SPLINE
SPL {X  -123.821, Y  +785.537, Z    +0.000, E1   -64.536, E3 +53300.374}
SPL {X  -153.467, Y  +737.853, Z    +0.000, E1   -51.757, E3 +53302.688}
SPL {X  -162.176, Y  +709.248, Z    +0.000, E1   -35.773, E3 +53301.714}
SPL {X  -164.888, Y  +691.368, Z    +0.000, E1   -20.174, E3 +53300.151}
SPL {X  -165.597, Y  +679.703, Z    +0.000, E1    -7.645, E3 +53300.327}
SPL {X  -165.650, Y  +673.520, Z    +0.000, E1    -0.048, E3 +53299.278}
SPL {X  -165.650, Y  +671.692, Z    +0.000, E1    +4.450, E3 +53298.845}
SPL {X  -165.650, Y  +667.743, Z    +0.000, E1   +15.617, E3 +53298.763}
SPL {X  -165.650, Y  +661.459, Z    +0.000, E1   +33.218, E3 +53298.343}
SPL {X  -165.650, Y  +653.296, Z    +0.000, E1   +51.333, E3 +53297.899}
SPL {X  -165.650, Y  +642.000, Z    +0.000, E1   +65.561, E3 +53297.111}
SPL {X  -165.650, Y  +619.979, Z    +0.000, E1   +79.465, E3 +53293.117}
SPL {X  -165.650, Y  +584.722, Z    +0.000, E1   +79.551, E3 +53302.408}
SPL {X  -165.650, Y  +560.326, Z    +0.000, E1   +78.360, E3 +53312.131}
SPL {X  -158.840, Y  +331.491, Z    +0.000, E1   +77.462, E3 +53394.706}
ENDSPLINE

SPLINE
SPL {X  -159.893, Y  +335.208, Z    +0.000, E1   +75.483, E3 +53415.441}
ENDSPLINE

SPLINE
SPL {X  -156.487, Y  +324.170, Z    +0.000, E1   +75.150, E3 +53424.822}
SPL {X  -142.256, Y  +293.629, Z    +0.000, E1   +77.020, E3 +53419.922}
ENDSPLINE

SPLINE
SPL {X  -142.811, Y  +294.566, Z    +0.000, E1   +75.668, E3 +53431.884}
ENDSPLINE

SPLINE
SPL {X  -141.646, Y  +292.615, Z    +0.000, E1   +74.702, E3 +53440.978}
SPL {X  -140.419, Y  +290.622, Z    +0.000, E1   +73.705, E3 +53449.821}
SPL {X  -136.008, Y  +283.940, Z    +0.000, E1   +73.594, E3 +53453.940}
SPL {X  -132.748, Y  +279.415, Z    +0.000, E1   +73.006, E3 +53459.996}
SPL {X  -129.007, Y  +274.590, Z    +0.000, E1   +72.484, E3 +53465.345}
SPL {X  -124.646, Y  +269.397, Z    +0.000, E1   +72.041, E3 +53470.093}
SPL {X  -111.023, Y  +255.562, Z    +0.000, E1   +75.772, E3 +53461.874}
SPL {X   -52.752, Y  +221.474, Z    +0.000, E1   +59.157, E3 +53591.126}
SPL {X   -49.901, Y  +220.545, Z    +0.000, E1   +56.696, E3 +53677.518}
ENDSPLINE

SPLINE
SPL {X  -127.117, Y  +272.287, Z    +0.000, E1   +62.713, E3 +53823.811}
SPL {X  -152.442, Y  +313.682, Z    +0.000, E1   +51.943, E3 +53828.043}
SPL {X  -159.925, Y  +335.326, Z    +0.000, E1   +41.361, E3 +53827.985}
SPL {X  -163.450, Y  +351.595, Z    +0.000, E1   +29.785, E3 +53827.096}
SPL {X  -165.127, Y  +365.342, Z    +0.000, E1   +17.250, E3 +53827.076}
SPL {X  -165.640, Y  +376.693, Z    +0.000, E1    +4.721, E3 +53826.649}
SPL {X  -165.650, Y  +380.500, Z    +0.000, E1    -0.000, E3 +53825.800}
SPL {X  -165.650, Y  +383.262, Z    +0.000, E1    -6.645, E3 +53825.329}
SPL {X  -165.650, Y  +388.390, Z    +0.000, E1   -21.508, E3 +53825.117}
SPL {X  -165.650, Y  +393.439, Z    +0.000, E1   -35.398, E3 +53824.685}
SPL {X  -165.650, Y  +400.610, Z    +0.000, E1   -50.510, E3 +53824.422}
SPL {X  -165.650, Y  +414.376, Z    +0.000, E1   -68.098, E3 +53822.456}
SPL {X  -165.650, Y  +468.582, Z    +0.000, E1   -78.237, E3 +53831.226}
SPL {X  -158.306, Y  +724.277, Z    +0.000, E1   -77.461, E3 +53921.667}
ENDSPLINE

SPLINE
SPL {X  -160.145, Y  +717.851, Z    +0.000, E1   -75.386, E3 +53942.181}
ENDSPLINE

SPLINE
SPL {X  -157.156, Y  +727.862, Z    +0.000, E1   -75.175, E3 +53949.653}
SPL {X  -154.068, Y  +736.353, Z    +0.000, E1   -74.906, E3 +53956.828}
SPL {X  -149.738, Y  +746.340, Z    +0.000, E1   -74.451, E3 +53966.515}
SPL {X  -145.204, Y  +755.223, Z    +0.000, E1   -74.188, E3 +53973.242}
SPL {X  -142.724, Y  +759.583, Z    +0.000, E1   -73.634, E3 +53980.061}
SPL {X  -138.277, Y  +766.711, Z    +0.000, E1   -73.303, E3 +53986.192}
SPL {X  -134.662, Y  +771.969, Z    +0.000, E1   -72.884, E3 +53991.634}
SPL {X  -131.459, Y  +776.289, Z    +0.000, E1   -72.475, E3 +53996.301}
SPL {X  -128.771, Y  +779.702, Z    +0.000, E1   -71.875, E3 +54001.248}
SPL {X  -125.267, Y  +783.889, Z    +0.000, E1   -71.674, E3 +54004.360}
SPL {X  -119.086, Y  +790.645, Z    +0.000, E1   -72.931, E3 +54002.647}
SPL {X   -51.449, Y  +832.958, Z    +0.000, E1   -57.230, E3 +54160.167}
ENDSPLINE

SPLINE
SPL {X  -123.821, Y  +785.537, Z    +0.000, E1   -64.536, E3 +54361.912}
SPL {X  -153.467, Y  +737.853, Z    +0.000, E1   -51.757, E3 +54364.227}
SPL {X  -162.176, Y  +709.248, Z    +0.000, E1   -35.773, E3 +54363.252}
SPL {X  -164.888, Y  +691.368, Z    +0.000, E1   -20.174, E3 +54361.690}
SPL {X  -165.597, Y  +679.703, Z    +0.000, E1    -7.645, E3 +54361.865}
SPL {X  -165.650, Y  +673.520, Z    +0.000, E1    -0.048, E3 +54360.817}
SPL {X  -165.650, Y  +671.692, Z    +0.000, E1    +4.450, E3 +54360.383}
SPL {X  -165.650, Y  +667.743, Z    +0.000, E1   +15.617, E3 +54360.301}
SPL {X  -165.650, Y  +662.891, Z    +0.000, E1   +29.740, E3 +54359.819}
SPL {X  -165.650, Y  +655.319, Z    +0.000, E1   +47.265, E3 +54359.668}
SPL {X  -165.650, Y  +642.000, Z    +0.000, E1   +65.561, E3 +54358.649}
SPL {X  -165.650, Y  +619.979, Z    +0.000, E1   +79.465, E3 +54354.656}
SPL {X  -165.650, Y  +569.632, Z    +0.000, E1   +78.783, E3 +54369.935}
SPL {X  -160.258, Y  +336.579, Z    +0.000, E1   +78.314, E3 +54445.191}
SPL {X  -159.618, Y  +334.207, Z    +0.000, E1   +75.622, E3 +54476.005}
SPL {X  -156.487, Y  +324.170, Z    +0.000, E1   +75.150, E3 +54486.360}
SPL {X  -142.256, Y  +293.629, Z    +0.000, E1   +77.020, E3 +54481.460}
ENDSPLINE

SPLINE
SPL {X  -142.811, Y  +294.566, Z    +0.000, E1   +75.668, E3 +54493.422}
ENDSPLINE

SPLINE
SPL {X  -141.646, Y  +292.615, Z    +0.000, E1   +74.702, E3 +54502.516}
SPL {X  -140.419, Y  +290.622, Z    +0.000, E1   +73.705, E3 +54511.359}
SPL {X  -136.008, Y  +283.940, Z    +0.000, E1   +73.594, E3 +54515.478}
SPL {X  -132.748, Y  +279.415, Z    +0.000, E1   +73.006, E3 +54521.534}
SPL {X  -129.007, Y  +274.590, Z    +0.000, E1   +72.484, E3 +54526.883}
SPL {X  -125.914, Y  +270.864, Z    +0.000, E1   +72.144, E3 +54530.375}
SPL {X  -123.729, Y  +268.359, Z    +0.000, E1   +71.932, E3 +54532.547}
SPL {X  -111.023, Y  +255.562, Z    +0.000, E1   +75.772, E3 +54523.413}
SPL {X   -49.289, Y  +220.353, Z    +0.000, E1   +56.690, E3 +54716.128}
ENDSPLINE

SPLINE
SPL {X  -127.117, Y  +272.287, Z    +0.000, E1   +62.713, E3 +54885.350}
SPL {X  -152.442, Y  +313.682, Z    +0.000, E1   +51.943, E3 +54889.581}
SPL {X  -159.925, Y  +335.326, Z    +0.000, E1   +41.361, E3 +54889.523}
SPL {X  -163.450, Y  +351.595, Z    +0.000, E1   +29.785, E3 +54888.635}
SPL {X  -165.127, Y  +365.342, Z    +0.000, E1   +17.250, E3 +54888.615}
SPL {X  -165.640, Y  +376.693, Z    +0.000, E1    +4.721, E3 +54888.188}
SPL {X  -165.650, Y  +380.500, Z    +0.000, E1    -0.000, E3 +54887.339}
SPL {X  -165.650, Y  +382.123, Z    +0.000, E1    -3.912, E3 +54886.966}
SPL {X  -165.650, Y  +387.069, Z    +0.000, E1   -17.420, E3 +54886.677}
SPL {X  -165.650, Y  +393.439, Z    +0.000, E1   -35.398, E3 +54886.223}
SPL {X  -165.650, Y  +400.610, Z    +0.000, E1   -50.510, E3 +54885.961}
SPL {X  -165.650, Y  +414.376, Z    +0.000, E1   -68.098, E3 +54883.994}
SPL {X  -165.650, Y  +468.582, Z    +0.000, E1   -78.237, E3 +54892.765}
SPL {X  -160.244, Y  +717.475, Z    +0.000, E1   -78.917, E3 +54965.322}
SPL {X  -159.651, Y  +719.676, Z    +0.000, E1   -75.661, E3 +55001.709}
SPL {X  -157.156, Y  +727.862, Z    +0.000, E1   -75.175, E3 +55011.191}
SPL {X  -152.814, Y  +739.436, Z    +0.000, E1   -74.813, E3 +55021.045}
SPL {X  -148.754, Y  +748.385, Z    +0.000, E1   -74.281, E3 +55030.487}
SPL {X  -144.163, Y  +757.090, Z    +0.000, E1   -74.033, E3 +55037.146}
SPL {X  -139.284, Y  +765.165, Z    +0.000, E1   -73.322, E3 +55046.841}
SPL {X  -134.662, Y  +771.969, Z    +0.000, E1   -72.884, E3 +55053.173}
SPL {X  -131.459, Y  +776.289, Z    +0.000, E1   -72.475, E3 +55057.840}
SPL {X  -128.771, Y  +779.702, Z    +0.000, E1   -71.875, E3 +55062.786}
SPL {X  -124.506, Y  +784.762, Z    +0.000, E1   -71.815, E3 +55065.675}
SPL {X  -112.958, Y  +796.663, Z    +0.000, E1   -74.119, E3 +55062.378}
SPL {X   -54.274, Y  +832.006, Z    +0.000, E1   -58.502, E3 +55194.398}
SPL {X   -50.797, Y  +833.169, Z    +0.000, E1   -57.000, E3 +55289.747}
ENDSPLINE

SPLINE
SPL {X  -113.713, Y  +795.955, Z    +0.000, E1   -65.735, E3 +55420.624}
SPL {X  -131.116, Y  +776.736, Z    +0.000, E1   -63.149, E3 +55425.154}
SPL {X  -153.467, Y  +737.853, Z    +0.000, E1   -51.757, E3 +55425.765}
SPL {X  -162.176, Y  +709.248, Z    +0.000, E1   -35.773, E3 +55424.791}
SPL {X  -164.888, Y  +691.368, Z    +0.000, E1   -20.174, E3 +55423.228}
SPL {X  -165.597, Y  +679.703, Z    +0.000, E1    -7.645, E3 +55423.403}
SPL {X  -165.650, Y  +673.520, Z    +0.000, E1    -0.048, E3 +55422.355}
SPL {X  -165.650, Y  +671.692, Z    +0.000, E1    +4.450, E3 +55421.922}
SPL {X  -165.650, Y  +667.743, Z    +0.000, E1   +15.617, E3 +55421.840}
SPL {X  -165.650, Y  +662.891, Z    +0.000, E1   +29.740, E3 +55421.358}
SPL {X  -165.650, Y  +655.319, Z    +0.000, E1   +47.265, E3 +55421.206}
SPL {X  -165.650, Y  +642.000, Z    +0.000, E1   +65.561, E3 +55420.188}
SPL {X  -165.650, Y  +619.979, Z    +0.000, E1   +79.465, E3 +55416.194}
SPL {X  -165.650, Y  +569.632, Z    +0.000, E1   +78.783, E3 +55431.473}
SPL {X  -158.840, Y  +331.491, Z    +0.000, E1   +77.462, E3 +55517.783}
ENDSPLINE

SPLINE
SPL {X  -159.893, Y  +335.208, Z    +0.000, E1   +75.483, E3 +55538.518}
ENDSPLINE

SPLINE
SPL {X  -156.487, Y  +324.170, Z    +0.000, E1   +75.150, E3 +55547.899}
SPL {X  -142.256, Y  +293.629, Z    +0.000, E1   +77.020, E3 +55542.999}
ENDSPLINE

SPLINE
SPL {X  -142.811, Y  +294.566, Z    +0.000, E1   +75.668, E3 +55554.961}
ENDSPLINE

SPLINE
SPL {X  -141.646, Y  +292.615, Z    +0.000, E1   +74.702, E3 +55564.055}
SPL {X  -140.419, Y  +290.622, Z    +0.000, E1   +73.705, E3 +55572.898}
SPL {X  -135.839, Y  +283.697, Z    +0.000, E1   +73.388, E3 +55578.636}
SPL {X  -131.336, Y  +277.551, Z    +0.000, E1   +72.879, E3 +55584.888}
SPL {X  -126.848, Y  +271.966, Z    +0.000, E1   +72.322, E3 +55590.617}
SPL {X  -123.729, Y  +268.359, Z    +0.000, E1   +71.932, E3 +55594.085}
SPL {X  -111.023, Y  +255.562, Z    +0.000, E1   +75.772, E3 +55584.951}
SPL {X   -52.752, Y  +221.474, Z    +0.000, E1   +59.157, E3 +55714.203}
SPL {X   -49.901, Y  +220.545, Z    +0.000, E1   +56.696, E3 +55800.595}
ENDSPLINE

SPLINE
SPL {X  -127.117, Y  +272.287, Z    +0.000, E1   +62.713, E3 +55946.888}
SPL {X  -152.442, Y  +313.682, Z    +0.000, E1   +51.943, E3 +55951.120}
SPL {X  -162.319, Y  +345.447, Z    +0.000, E1   +34.671, E3 +55950.545}
SPL {X  -165.127, Y  +365.342, Z    +0.000, E1   +17.250, E3 +55950.153}
SPL {X  -165.640, Y  +376.693, Z    +0.000, E1    +4.721, E3 +55949.726}
SPL {X  -165.650, Y  +380.500, Z    +0.000, E1    -0.000, E3 +55948.877}
SPL {X  -165.650, Y  +383.262, Z    +0.000, E1    -6.645, E3 +55948.406}
SPL {X  -165.650, Y  +388.390, Z    +0.000, E1   -21.508, E3 +55948.194}
SPL {X  -165.650, Y  +393.439, Z    +0.000, E1   -35.398, E3 +55947.762}
SPL {X  -165.650, Y  +400.610, Z    +0.000, E1   -50.510, E3 +55947.499}
SPL {X  -165.650, Y  +414.376, Z    +0.000, E1   -68.098, E3 +55945.533}
SPL {X  -165.650, Y  +468.582, Z    +0.000, E1   -78.237, E3 +55954.303}
SPL {X  -158.306, Y  +724.277, Z    +0.000, E1   -77.461, E3 +56044.744}
ENDSPLINE

SPLINE
SPL {X  -160.145, Y  +717.851, Z    +0.000, E1   -75.386, E3 +56065.258}
ENDSPLINE

SPLINE
SPL {X  -157.156, Y  +727.862, Z    +0.000, E1   -75.175, E3 +56072.730}
SPL {X  -152.814, Y  +739.436, Z    +0.000, E1   -74.813, E3 +56082.583}
SPL {X  -148.754, Y  +748.385, Z    +0.000, E1   -74.281, E3 +56092.026}
SPL {X  -144.163, Y  +757.090, Z    +0.000, E1   -74.033, E3 +56098.685}
SPL {X  -139.284, Y  +765.165, Z    +0.000, E1   -73.322, E3 +56108.379}
SPL {X  -134.662, Y  +771.969, Z    +0.000, E1   -72.884, E3 +56114.711}
SPL {X  -131.459, Y  +776.289, Z    +0.000, E1   -72.475, E3 +56119.378}
SPL {X  -127.605, Y  +781.126, Z    +0.000, E1   -71.922, E3 +56124.822}
SPL {X  -124.773, Y  +784.457, Z    +0.000, E1   -71.383, E3 +56128.870}
SPL {X  -119.086, Y  +790.645, Z    +0.000, E1   -72.931, E3 +56125.724}
SPL {X   -51.449, Y  +832.958, Z    +0.000, E1   -57.230, E3 +56283.244}
ENDSPLINE

SPLINE
SPL {X  -123.821, Y  +785.537, Z    +0.000, E1   -64.536, E3 +56484.989}
SPL {X  -153.467, Y  +737.853, Z    +0.000, E1   -51.757, E3 +56487.304}
SPL {X  -162.176, Y  +709.248, Z    +0.000, E1   -35.773, E3 +56486.329}
SPL {X  -164.888, Y  +691.368, Z    +0.000, E1   -20.174, E3 +56484.767}
SPL {X  -165.597, Y  +679.703, Z    +0.000, E1    -7.645, E3 +56484.942}
SPL {X  -165.650, Y  +673.520, Z    +0.000, E1    -0.048, E3 +56483.894}
SPL {X  -165.650, Y  +671.692, Z    +0.000, E1    +4.450, E3 +56483.460}
SPL {X  -165.650, Y  +667.743, Z    +0.000, E1   +15.617, E3 +56483.378}
SPL {X  -165.650, Y  +661.459, Z    +0.000, E1   +33.218, E3 +56482.959}
SPL {X  -165.650, Y  +653.296, Z    +0.000, E1   +51.333, E3 +56482.514}
SPL {X  -165.650, Y  +642.000, Z    +0.000, E1   +65.561, E3 +56481.726}
SPL {X  -165.650, Y  +619.979, Z    +0.000, E1   +79.465, E3 +56477.733}
SPL {X  -165.650, Y  +584.722, Z    +0.000, E1   +79.551, E3 +56487.023}
SPL {X  -165.650, Y  +560.326, Z    +0.000, E1   +78.360, E3 +56496.746}
SPL {X  -158.840, Y  +331.491, Z    +0.000, E1   +77.462, E3 +56579.322}
ENDSPLINE

SPLINE
SPL {X  -159.893, Y  +335.208, Z    +0.000, E1   +75.483, E3 +56600.056}
ENDSPLINE

SPLINE
SPL {X  -156.487, Y  +324.170, Z    +0.000, E1   +75.150, E3 +56609.437}
SPL {X  -142.256, Y  +293.629, Z    +0.000, E1   +77.020, E3 +56604.537}
ENDSPLINE

SPLINE
SPL {X  -142.811, Y  +294.566, Z    +0.000, E1   +75.668, E3 +56616.499}
ENDSPLINE

SPLINE
SPL {X  -141.646, Y  +292.615, Z    +0.000, E1   +74.702, E3 +56625.593}
SPL {X  -140.419, Y  +290.622, Z    +0.000, E1   +73.705, E3 +56634.436}
SPL {X  -136.008, Y  +283.940, Z    +0.000, E1   +73.594, E3 +56638.555}
SPL {X  -132.748, Y  +279.415, Z    +0.000, E1   +73.006, E3 +56644.611}
SPL {X  -129.007, Y  +274.590, Z    +0.000, E1   +72.484, E3 +56649.960}
SPL {X  -124.646, Y  +269.397, Z    +0.000, E1   +72.041, E3 +56654.708}
SPL {X  -111.023, Y  +255.562, Z    +0.000, E1   +75.772, E3 +56646.490}
SPL {X   -52.752, Y  +221.474, Z    +0.000, E1   +59.157, E3 +56775.741}
SPL {X   -49.901, Y  +220.545, Z    +0.000, E1   +56.696, E3 +56862.134}
ENDSPLINE

SPLINE
SPL {X  -127.117, Y  +272.287, Z    +0.000, E1   +62.713, E3 +57008.427}
SPL {X  -152.442, Y  +313.682, Z    +0.000, E1   +51.943, E3 +57012.658}
SPL {X  -159.925, Y  +335.326, Z    +0.000, E1   +41.361, E3 +57012.600}
SPL {X  -163.450, Y  +351.595, Z    +0.000, E1   +29.785, E3 +57011.712}
SPL {X  -165.127, Y  +365.342, Z    +0.000, E1   +17.250, E3 +57011.692}
SPL {X  -165.640, Y  +376.693, Z    +0.000, E1    +4.721, E3 +57011.265}
SPL {X  -165.650, Y  +380.500, Z    +0.000, E1    -0.000, E3 +57010.416}
SPL {X  -165.650, Y  +383.262, Z    +0.000, E1    -6.645, E3 +57009.945}
SPL {X  -165.650, Y  +388.390, Z    +0.000, E1   -21.508, E3 +57009.733}
SPL {X  -165.650, Y  +393.439, Z    +0.000, E1   -35.398, E3 +57009.300}
SPL {X  -165.650, Y  +400.610, Z    +0.000, E1   -50.510, E3 +57009.038}
SPL {X  -165.650, Y  +414.376, Z    +0.000, E1   -68.098, E3 +57007.071}
SPL {X  -165.650, Y  +468.582, Z    +0.000, E1   -78.237, E3 +57015.841}
SPL {X  -158.306, Y  +724.277, Z    +0.000, E1   -77.461, E3 +57106.283}
ENDSPLINE

SPLINE
SPL {X  -160.145, Y  +717.851, Z    +0.000, E1   -75.386, E3 +57126.796}
ENDSPLINE

SPLINE
SPL {X  -157.156, Y  +727.862, Z    +0.000, E1   -75.175, E3 +57134.268}
SPL {X  -152.814, Y  +739.436, Z    +0.000, E1   -74.813, E3 +57144.122}
SPL {X  -147.104, Y  +751.659, Z    +0.000, E1   -74.255, E3 +57155.566}
SPL {X  -141.453, Y  +761.704, Z    +0.000, E1   -73.638, E3 +57165.779}
SPL {X  -135.914, Y  +770.196, Z    +0.000, E1   -72.974, E3 +57174.841}
SPL {X  -131.459, Y  +776.289, Z    +0.000, E1   -72.475, E3 +57180.917}
SPL {X  -127.605, Y  +781.126, Z    +0.000, E1   -71.922, E3 +57186.361}
SPL {X  -124.773, Y  +784.457, Z    +0.000, E1   -71.383, E3 +57190.408}
SPL {X  -119.086, Y  +790.645, Z    +0.000, E1   -72.931, E3 +57187.262}
SPL {X   -51.449, Y  +832.958, Z    +0.000, E1   -57.230, E3 +57344.782}
ENDSPLINE

SPLINE
SPL {X  -113.713, Y  +795.955, Z    +0.000, E1   -65.735, E3 +57543.701}
SPL {X  -131.116, Y  +776.736, Z    +0.000, E1   -63.149, E3 +57548.231}
SPL {X  -153.467, Y  +737.853, Z    +0.000, E1   -51.757, E3 +57548.842}
SPL {X  -161.000, Y  +714.475, Z    +0.000, E1   -39.424, E3 +57548.315}
SPL {X  -164.534, Y  +694.695, Z    +0.000, E1   -23.511, E3 +57546.605}
SPL {X  -165.597, Y  +679.703, Z    +0.000, E1    -7.645, E3 +57546.480}
SPL {X  -165.650, Y  +673.520, Z    +0.000, E1    -0.048, E3 +57545.432}
SPL {X  -165.650, Y  +671.692, Z    +0.000, E1    +4.450, E3 +57544.999}
SPL {X  -165.650, Y  +667.743, Z    +0.000, E1   +15.617, E3 +57544.917}
SPL {X  -165.650, Y  +661.459, Z    +0.000, E1   +33.218, E3 +57544.497}
SPL {X  -165.650, Y  +650.834, Z    +0.000, E1   +55.143, E3 +57543.885}
SPL {X  -165.650, Y  +639.785, Z    +0.000, E1   +67.512, E3 +57543.102}
SPL {X  -165.650, Y  +619.979, Z    +0.000, E1   +79.465, E3 +57539.271}
SPL {X  -165.650, Y  +584.722, Z    +0.000, E1   +79.551, E3 +57548.562}
SPL {X  -165.650, Y  +560.326, Z    +0.000, E1   +78.360, E3 +57558.284}
SPL {X  -160.258, Y  +336.579, Z    +0.000, E1   +78.314, E3 +57629.806}
SPL {X  -159.618, Y  +334.207, Z    +0.000, E1   +75.622, E3 +57660.620}
SPL {X  -156.487, Y  +324.170, Z    +0.000, E1   +75.150, E3 +57670.976}
SPL {X  -142.256, Y  +293.629, Z    +0.000, E1   +77.020, E3 +57666.076}
ENDSPLINE

SPLINE
SPL {X  -142.811, Y  +294.566, Z    +0.000, E1   +75.668, E3 +57678.038}
ENDSPLINE

SPLINE
SPL {X  -141.646, Y  +292.615, Z    +0.000, E1   +74.702, E3 +57687.131}
SPL {X  -140.419, Y  +290.622, Z    +0.000, E1   +73.705, E3 +57695.975}
SPL {X  -135.839, Y  +283.697, Z    +0.000, E1   +73.388, E3 +57701.713}
SPL {X  -131.903, Y  +278.292, Z    +0.000, E1   +73.096, E3 +57706.202}
SPL {X  -129.007, Y  +274.590, Z    +0.000, E1   +72.484, E3 +57711.498}
SPL {X  -124.646, Y  +269.397, Z    +0.000, E1   +72.041, E3 +57716.247}
SPL {X  -111.023, Y  +255.562, Z    +0.000, E1   +75.772, E3 +57708.028}
SPL {X   -49.289, Y  +220.353, Z    +0.000, E1   +56.690, E3 +57900.743}
ENDSPLINE

SPLINE
SPL {X  -127.117, Y  +272.287, Z    +0.000, E1   +62.713, E3 +58069.965}
SPL {X  -152.442, Y  +313.682, Z    +0.000, E1   +51.943, E3 +58074.197}
SPL {X  -159.925, Y  +335.326, Z    +0.000, E1   +41.361, E3 +58074.139}
SPL {X  -163.450, Y  +351.595, Z    +0.000, E1   +29.785, E3 +58073.250}
SPL {X  -165.127, Y  +365.342, Z    +0.000, E1   +17.250, E3 +58073.230}
SPL {X  -165.640, Y  +376.693, Z    +0.000, E1    +4.721, E3 +58072.803}
SPL {X  -165.650, Y  +380.500, Z    +0.000, E1    -0.000, E3 +58071.954}
SPL {X  -165.650, Y  +382.123, Z    +0.000, E1    -3.912, E3 +58071.581}
SPL {X  -165.650, Y  +387.069, Z    +0.000, E1   -17.420, E3 +58071.293}
SPL {X  -165.650, Y  +393.439, Z    +0.000, E1   -35.398, E3 +58070.839}
SPL {X  -165.650, Y  +400.610, Z    +0.000, E1   -50.510, E3 +58070.576}
SPL {X  -165.650, Y  +414.376, Z    +0.000, E1   -68.098, E3 +58068.610}
SPL {X  -165.650, Y  +468.582, Z    +0.000, E1   -78.237, E3 +58077.380}
SPL {X  -158.306, Y  +724.277, Z    +0.000, E1   -77.461, E3 +58167.821}
ENDSPLINE

SPLINE
SPL {X  -160.145, Y  +717.851, Z    +0.000, E1   -75.386, E3 +58188.335}
ENDSPLINE

SPLINE
SPL {X  -157.156, Y  +727.862, Z    +0.000, E1   -75.175, E3 +58195.807}
SPL {X  -154.068, Y  +736.353, Z    +0.000, E1   -74.906, E3 +58202.981}
SPL {X  -149.738, Y  +746.340, Z    +0.000, E1   -74.451, E3 +58212.669}
SPL {X  -145.204, Y  +755.223, Z    +0.000, E1   -74.188, E3 +58219.395}
SPL {X  -142.724, Y  +759.583, Z    +0.000, E1   -73.634, E3 +58226.215}
SPL {X  -138.277, Y  +766.711, Z    +0.000, E1   -73.303, E3 +58232.346}
SPL {X  -134.662, Y  +771.969, Z    +0.000, E1   -72.884, E3 +58237.788}
SPL {X  -131.459, Y  +776.289, Z    +0.000, E1   -72.475, E3 +58242.455}
SPL {X  -128.771, Y  +779.702, Z    +0.000, E1   -71.875, E3 +58247.402}
SPL {X  -124.506, Y  +784.762, Z    +0.000, E1   -71.815, E3 +58250.290}
SPL {X  -112.958, Y  +796.663, Z    +0.000, E1   -74.119, E3 +58246.994}
SPL {X   -51.449, Y  +832.958, Z    +0.000, E1   -57.230, E3 +58406.321}
ENDSPLINE

SPLINE
SPL {X  -123.821, Y  +785.537, Z    +0.000, E1   -64.536, E3 +58608.066}
SPL {X  -153.467, Y  +737.853, Z    +0.000, E1   -51.757, E3 +58610.381}
SPL {X  -161.000, Y  +714.475, Z    +0.000, E1   -39.424, E3 +58609.853}
SPL {X  -164.534, Y  +694.695, Z    +0.000, E1   -23.511, E3 +58608.143}
SPL {X  -165.597, Y  +679.703, Z    +0.000, E1    -7.645, E3 +58608.019}
SPL {X  -165.650, Y  +673.520, Z    +0.000, E1    -0.048, E3 +58606.971}
SPL {X  -165.650, Y  +671.692, Z    +0.000, E1    +4.450, E3 +58606.537}
SPL {X  -165.650, Y  +667.743, Z    +0.000, E1   +15.617, E3 +58606.455}
SPL {X  -165.650, Y  +662.891, Z    +0.000, E1   +29.740, E3 +58605.973}
SPL {X  -165.650, Y  +655.319, Z    +0.000, E1   +47.265, E3 +58605.822}
SPL {X  -165.650, Y  +642.000, Z    +0.000, E1   +65.561, E3 +58604.803}
SPL {X  -165.650, Y  +619.979, Z    +0.000, E1   +79.465, E3 +58600.810}
SPL {X  -165.650, Y  +569.632, Z    +0.000, E1   +78.783, E3 +58616.088}
SPL {X  -158.840, Y  +331.491, Z    +0.000, E1   +77.462, E3 +58702.398}
ENDSPLINE

SPLINE
SPL {X  -159.893, Y  +335.208, Z    +0.000, E1   +75.483, E3 +58723.133}
ENDSPLINE

SPLINE
SPL {X  -156.487, Y  +324.170, Z    +0.000, E1   +75.150, E3 +58732.514}
SPL {X  -142.256, Y  +293.629, Z    +0.000, E1   +77.020, E3 +58727.614}
ENDSPLINE

SPLINE
SPL {X  -142.811, Y  +294.566, Z    +0.000, E1   +75.668, E3 +58739.576}
ENDSPLINE

SPLINE
SPL {X  -141.646, Y  +292.615, Z    +0.000, E1   +74.702, E3 +58748.670}
SPL {X  -140.419, Y  +290.622, Z    +0.000, E1   +73.705, E3 +58757.513}
SPL {X  -136.008, Y  +283.940, Z    +0.000, E1   +73.594, E3 +58761.632}
SPL {X  -132.748, Y  +279.415, Z    +0.000, E1   +73.006, E3 +58767.688}
SPL {X  -129.007, Y  +274.590, Z    +0.000, E1   +72.484, E3 +58773.037}
SPL {X  -125.914, Y  +270.864, Z    +0.000, E1   +72.144, E3 +58776.528}
SPL {X  -123.729, Y  +268.359, Z    +0.000, E1   +71.932, E3 +58778.701}
SPL {X  -111.023, Y  +255.562, Z    +0.000, E1   +75.772, E3 +58769.567}
SPL {X   -52.752, Y  +221.474, Z    +0.000, E1   +59.157, E3 +58898.818}
SPL {X   -49.901, Y  +220.545, Z    +0.000, E1   +56.696, E3 +58985.211}
ENDSPLINE

SPLINE
SPL {X  -127.117, Y  +272.287, Z    +0.000, E1   +62.713, E3 +59131.503}
SPL {X  -152.442, Y  +313.682, Z    +0.000, E1   +51.943, E3 +59135.735}
SPL {X  -162.319, Y  +345.447, Z    +0.000, E1   +34.671, E3 +59135.161}
SPL {X  -165.127, Y  +365.342, Z    +0.000, E1   +17.250, E3 +59134.769}
SPL {X  -165.640, Y  +376.693, Z    +0.000, E1    +4.721, E3 +59134.342}
SPL {X  -165.650, Y  +380.500, Z    +0.000, E1    -0.000, E3 +59133.493}
SPL {X  -165.650, Y  +382.123, Z    +0.000, E1    -3.912, E3 +59133.120}
SPL {X  -165.650, Y  +387.069, Z    +0.000, E1   -17.420, E3 +59132.831}
SPL {X  -165.650, Y  +393.439, Z    +0.000, E1   -35.398, E3 +59132.377}
SPL {X  -165.650, Y  +400.610, Z    +0.000, E1   -50.510, E3 +59132.115}
SPL {X  -165.650, Y  +414.376, Z    +0.000, E1   -68.098, E3 +59130.148}
SPL {X  -165.650, Y  +468.582, Z    +0.000, E1   -78.237, E3 +59138.918}
SPL {X  -158.306, Y  +724.277, Z    +0.000, E1   -77.461, E3 +59229.360}
ENDSPLINE

SPLINE
SPL {X  -160.145, Y  +717.851, Z    +0.000, E1   -75.386, E3 +59249.873}
ENDSPLINE

SPLINE
SPL {X  -157.156, Y  +727.862, Z    +0.000, E1   -75.175, E3 +59257.345}
SPL {X  -154.068, Y  +736.353, Z    +0.000, E1   -74.906, E3 +59264.520}
SPL {X  -149.738, Y  +746.340, Z    +0.000, E1   -74.451, E3 +59274.208}
SPL {X  -144.163, Y  +757.090, Z    +0.000, E1   -74.033, E3 +59283.300}
SPL {X  -139.284, Y  +765.165, Z    +0.000, E1   -73.322, E3 +59292.995}
SPL {X  -134.662, Y  +771.969, Z    +0.000, E1   -72.884, E3 +59299.326}
SPL {X  -131.459, Y  +776.289, Z    +0.000, E1   -72.475, E3 +59303.994}
SPL {X  -127.605, Y  +781.126, Z    +0.000, E1   -71.922, E3 +59309.438}
SPL {X  -124.773, Y  +784.457, Z    +0.000, E1   -71.383, E3 +59313.485}
SPL {X  -119.086, Y  +790.645, Z    +0.000, E1   -72.931, E3 +59310.339}
SPL {X   -51.449, Y  +832.958, Z    +0.000, E1   -57.230, E3 +59467.859}
ENDSPLINE

SPLINE
SPL {X  -123.821, Y  +785.537, Z    +0.000, E1   -64.536, E3 +59669.604}
SPL {X  -153.467, Y  +737.853, Z    +0.000, E1   -51.757, E3 +59671.919}
SPL {X  -161.000, Y  +714.475, Z    +0.000, E1   -39.424, E3 +59671.392}
SPL {X  -164.534, Y  +694.695, Z    +0.000, E1   -23.511, E3 +59669.682}
SPL {X  -165.597, Y  +679.703, Z    +0.000, E1    -7.645, E3 +59669.557}
SPL {X  -165.650, Y  +673.520, Z    +0.000, E1    -0.048, E3 +59668.509}
SPL {X  -165.650, Y  +671.692, Z    +0.000, E1    +4.450, E3 +59668.076}
SPL {X  -165.650, Y  +667.743, Z    +0.000, E1   +15.617, E3 +59667.994}
SPL {X  -165.650, Y  +662.891, Z    +0.000, E1   +29.740, E3 +59667.511}
SPL {X  -165.650, Y  +655.319, Z    +0.000, E1   +47.265, E3 +59667.360}
SPL {X  -165.650, Y  +642.000, Z    +0.000, E1   +65.561, E3 +59666.341}
SPL {X  -165.650, Y  +619.979, Z    +0.000, E1   +79.465, E3 +59662.348}
SPL {X  -165.650, Y  +569.632, Z    +0.000, E1   +78.783, E3 +59677.627}
SPL {X  -160.258, Y  +336.579, Z    +0.000, E1   +78.314, E3 +59752.883}
SPL {X  -159.618, Y  +334.207, Z    +0.000, E1   +75.622, E3 +59783.697}
SPL {X  -156.487, Y  +324.170, Z    +0.000, E1   +75.150, E3 +59794.053}
SPL {X  -142.256, Y  +293.629, Z    +0.000, E1   +77.020, E3 +59789.152}
ENDSPLINE

SPLINE
SPL {X  -142.811, Y  +294.566, Z    +0.000, E1   +75.668, E3 +59801.115}
ENDSPLINE

SPLINE
SPL {X  -141.646, Y  +292.615, Z    +0.000, E1   +74.702, E3 +59810.208}
SPL {X  -140.419, Y  +290.622, Z    +0.000, E1   +73.705, E3 +59819.052}
SPL {X  -135.839, Y  +283.697, Z    +0.000, E1   +73.388, E3 +59824.790}
SPL {X  -131.336, Y  +277.551, Z    +0.000, E1   +72.879, E3 +59831.042}
SPL {X  -126.848, Y  +271.966, Z    +0.000, E1   +72.322, E3 +59836.770}
SPL {X  -123.729, Y  +268.359, Z    +0.000, E1   +71.932, E3 +59840.239}
SPL {X  -111.023, Y  +255.562, Z    +0.000, E1   +75.772, E3 +59831.105}
SPL {X   -49.289, Y  +220.353, Z    +0.000, E1   +56.690, E3 +60023.820}
ENDSPLINE

SPLINE
SPL {X  -127.117, Y  +272.287, Z    +0.000, E1   +62.713, E3 +60193.042}
SPL {X  -152.442, Y  +313.682, Z    +0.000, E1   +51.943, E3 +60197.274}
SPL {X  -159.925, Y  +335.326, Z    +0.000, E1   +41.361, E3 +60197.216}
SPL {X  -163.450, Y  +351.595, Z    +0.000, E1   +29.785, E3 +60196.327}
SPL {X  -165.127, Y  +365.342, Z    +0.000, E1   +17.250, E3 +60196.307}
SPL {X  -165.640, Y  +376.693, Z    +0.000, E1    +4.721, E3 +60195.880}
SPL {X  -165.650, Y  +380.500, Z    +0.000, E1    -0.000, E3 +60195.031}
SPL {X  -165.650, Y  +382.123, Z    +0.000, E1    -3.912, E3 +60194.658}
SPL {X  -165.650, Y  +387.069, Z    +0.000, E1   -17.420, E3 +60194.370}
SPL {X  -165.650, Y  +393.439, Z    +0.000, E1   -35.398, E3 +60193.915}
SPL {X  -165.650, Y  +400.610, Z    +0.000, E1   -50.510, E3 +60193.653}
SPL {X  -165.650, Y  +414.376, Z    +0.000, E1   -68.098, E3 +60191.687}
SPL {X  -165.650, Y  +468.582, Z    +0.000, E1   -78.237, E3 +60200.457}
SPL {X  -158.306, Y  +724.277, Z    +0.000, E1   -77.461, E3 +60290.898}
ENDSPLINE

SPLINE
SPL {X  -160.145, Y  +717.851, Z    +0.000, E1   -75.386, E3 +60311.412}
ENDSPLINE

SPLINE
SPL {X  -157.156, Y  +727.862, Z    +0.000, E1   -75.175, E3 +60318.884}
SPL {X  -154.068, Y  +736.353, Z    +0.000, E1   -74.906, E3 +60326.058}
SPL {X  -149.738, Y  +746.340, Z    +0.000, E1   -74.451, E3 +60335.746}
SPL {X  -145.204, Y  +755.223, Z    +0.000, E1   -74.188, E3 +60342.472}
SPL {X  -142.724, Y  +759.583, Z    +0.000, E1   -73.634, E3 +60349.292}
SPL {X  -138.277, Y  +766.711, Z    +0.000, E1   -73.303, E3 +60355.422}
SPL {X  -134.662, Y  +771.969, Z    +0.000, E1   -72.884, E3 +60360.865}
SPL {X  -131.459, Y  +776.289, Z    +0.000, E1   -72.475, E3 +60365.532}
SPL {X  -128.771, Y  +779.702, Z    +0.000, E1   -71.875, E3 +60370.479}
SPL {X  -124.506, Y  +784.762, Z    +0.000, E1   -71.815, E3 +60373.367}
SPL {X  -112.958, Y  +796.663, Z    +0.000, E1   -74.119, E3 +60370.071}
SPL {X   -51.449, Y  +832.958, Z    +0.000, E1   -57.230, E3 +60529.398}
ENDSPLINE

SPLINE
SPL {X  -123.821, Y  +785.537, Z    +0.000, E1   -64.536, E3 +60731.143}
SPL {X  -153.467, Y  +737.853, Z    +0.000, E1   -51.757, E3 +60733.458}
SPL {X  -161.000, Y  +714.475, Z    +0.000, E1   -39.424, E3 +60732.930}
SPL {X  -164.534, Y  +694.695, Z    +0.000, E1   -23.511, E3 +60731.220}
SPL {X  -165.597, Y  +679.703, Z    +0.000, E1    -7.645, E3 +60731.096}
SPL {X  -165.650, Y  +673.520, Z    +0.000, E1    -0.048, E3 +60730.048}
SPL {X  -165.650, Y  +671.692, Z    +0.000, E1    +4.450, E3 +60729.614}
SPL {X  -165.650, Y  +667.743, Z    +0.000, E1   +15.617, E3 +60729.532}
SPL {X  -165.650, Y  +662.891, Z    +0.000, E1   +29.740, E3 +60729.050}
SPL {X  -165.650, Y  +655.319, Z    +0.000, E1   +47.265, E3 +60728.899}
SPL {X  -165.650, Y  +642.000, Z    +0.000, E1   +65.561, E3 +60727.880}
SPL {X  -165.650, Y  +619.979, Z    +0.000, E1   +79.465, E3 +60723.886}
SPL {X  -165.650, Y  +569.632, Z    +0.000, E1   +78.783, E3 +60739.165}
SPL {X  -160.258, Y  +336.579, Z    +0.000, E1   +78.314, E3 +60814.422}
SPL {X  -159.618, Y  +334.207, Z    +0.000, E1   +75.622, E3 +60845.235}
SPL {X  -156.487, Y  +324.170, Z    +0.000, E1   +75.150, E3 +60855.591}
SPL {X  -142.256, Y  +293.629, Z    +0.000, E1   +77.020, E3 +60850.691}
ENDSPLINE

SPLINE
SPL {X  -142.811, Y  +294.566, Z    +0.000, E1   +75.668, E3 +60862.653}
ENDSPLINE

SPLINE
SPL {X  -141.646, Y  +292.615, Z    +0.000, E1   +74.702, E3 +60871.747}
SPL {X  -140.419, Y  +290.622, Z    +0.000, E1   +73.705, E3 +60880.590}
SPL {X  -135.839, Y  +283.697, Z    +0.000, E1   +73.388, E3 +60886.328}
SPL {X  -131.336, Y  +277.551, Z    +0.000, E1   +72.879, E3 +60892.581}
SPL {X  -126.848, Y  +271.966, Z    +0.000, E1   +72.322, E3 +60898.309}
SPL {X  -123.729, Y  +268.359, Z    +0.000, E1   +71.932, E3 +60901.778}
SPL {X  -111.023, Y  +255.562, Z    +0.000, E1   +75.772, E3 +60892.644}
SPL {X   -49.289, Y  +220.353, Z    +0.000, E1   +56.690, E3 +61085.358}
ENDSPLINE

SPLINE
SPL {X  -127.117, Y  +272.287, Z    +0.000, E1   +62.713, E3 +61254.580}
SPL {X  -152.442, Y  +313.682, Z    +0.000, E1   +51.943, E3 +61258.812}
SPL {X  -159.925, Y  +335.326, Z    +0.000, E1   +41.361, E3 +61258.754}
SPL {X  -163.450, Y  +351.595, Z    +0.000, E1   +29.785, E3 +61257.865}
SPL {X  -165.127, Y  +365.342, Z    +0.000, E1   +17.250, E3 +61257.846}
SPL {X  -165.640, Y  +376.693, Z    +0.000, E1    +4.721, E3 +61257.419}
SPL {X  -165.650, Y  +380.500, Z    +0.000, E1    -0.000, E3 +61256.569}
SPL {X  -165.650, Y  +382.123, Z    +0.000, E1    -3.912, E3 +61256.197}
SPL {X  -165.650, Y  +387.069, Z    +0.000, E1   -17.420, E3 +61255.908}
SPL {X  -165.650, Y  +393.439, Z    +0.000, E1   -35.398, E3 +61255.454}
SPL {X  -165.650, Y  +402.896, Z    +0.000, E1   -54.480, E3 +61254.695}
SPL {X  -165.650, Y  +416.934, Z    +0.000, E1   -69.887, E3 +61253.161}
SPL {X  -165.650, Y  +459.729, Z    +0.000, E1   -78.035, E3 +61259.680}
SPL {X  -165.650, Y  +475.450, Z    +0.000, E1   -78.345, E3 +61263.794}
SPL {X  -160.244, Y  +717.475, Z    +0.000, E1   -78.917, E3 +61334.553}
SPL {X  -159.651, Y  +719.676, Z    +0.000, E1   -75.661, E3 +61370.940}
SPL {X  -157.156, Y  +727.862, Z    +0.000, E1   -75.175, E3 +61380.422}
SPL {X  -154.068, Y  +736.353, Z    +0.000, E1   -74.906, E3 +61387.597}
SPL {X  -149.738, Y  +746.340, Z    +0.000, E1   -74.451, E3 +61397.284}
SPL {X  -144.163, Y  +757.090, Z    +0.000, E1   -74.033, E3 +61406.377}
SPL {X  -140.473, Y  +763.291, Z    +0.000, E1   -73.478, E3 +61413.818}
SPL {X  -135.914, Y  +770.196, Z    +0.000, E1   -72.974, E3 +61420.995}
SPL {X  -131.459, Y  +776.289, Z    +0.000, E1   -72.475, E3 +61427.070}
SPL {X  -128.771, Y  +779.702, Z    +0.000, E1   -71.875, E3 +61432.017}
SPL {X  -124.506, Y  +784.762, Z    +0.000, E1   -71.815, E3 +61434.906}
SPL {X  -112.958, Y  +796.663, Z    +0.000, E1   -74.119, E3 +61431.609}
SPL {X   -51.449, Y  +832.958, Z    +0.000, E1   -57.230, E3 +61590.936}
ENDSPLINE

SPLINE
SPL {X  -123.821, Y  +785.537, Z    +0.000, E1   -64.536, E3 +61792.681}
SPL {X  -153.467, Y  +737.853, Z    +0.000, E1   -51.757, E3 +61794.996}
SPL {X  -161.000, Y  +714.475, Z    +0.000, E1   -39.424, E3 +61794.469}
SPL {X  -164.534, Y  +694.695, Z    +0.000, E1   -23.511, E3 +61792.759}
SPL {X  -165.597, Y  +679.703, Z    +0.000, E1    -7.645, E3 +61792.634}
SPL {X  -165.650, Y  +673.520, Z    +0.000, E1    -0.048, E3 +61791.586}
SPL {X  -165.650, Y  +671.692, Z    +0.000, E1    +4.450, E3 +61791.153}
SPL {X  -165.650, Y  +667.743, Z    +0.000, E1   +15.617, E3 +61791.070}
SPL {X  -165.650, Y  +662.891, Z    +0.000, E1   +29.740, E3 +61790.588}
SPL {X  -165.650, Y  +655.319, Z    +0.000, E1   +47.265, E3 +61790.437}
SPL {X  -165.650, Y  +642.000, Z    +0.000, E1   +65.561, E3 +61789.418}
SPL {X  -165.650, Y  +619.979, Z    +0.000, E1   +79.465, E3 +61785.425}
SPL {X  -165.650, Y  +569.632, Z    +0.000, E1   +78.783, E3 +61800.704}
SPL {X  -158.840, Y  +331.491, Z    +0.000, E1   +77.462, E3 +61887.014}
ENDSPLINE

SPLINE
SPL {X  -159.893, Y  +335.208, Z    +0.000, E1   +75.483, E3 +61907.748}
ENDSPLINE

SPLINE
SPL {X  -156.487, Y  +324.170, Z    +0.000, E1   +75.150, E3 +61917.130}
SPL {X  -142.256, Y  +293.629, Z    +0.000, E1   +77.020, E3 +61912.229}
ENDSPLINE

SPLINE
SPL {X  -142.811, Y  +294.566, Z    +0.000, E1   +75.668, E3 +61924.192}
ENDSPLINE

SPLINE
SPL {X  -141.646, Y  +292.615, Z    +0.000, E1   +74.702, E3 +61933.285}
SPL {X  -140.419, Y  +290.622, Z    +0.000, E1   +73.705, E3 +61942.129}
SPL {X  -135.839, Y  +283.697, Z    +0.000, E1   +73.388, E3 +61947.867}
SPL {X  -131.903, Y  +278.292, Z    +0.000, E1   +73.096, E3 +61952.356}
SPL {X  -129.007, Y  +274.590, Z    +0.000, E1   +72.484, E3 +61957.652}
SPL {X  -124.646, Y  +269.397, Z    +0.000, E1   +72.041, E3 +61962.400}
SPL {X  -111.023, Y  +255.562, Z    +0.000, E1   +75.772, E3 +61954.182}
SPL {X   -49.289, Y  +220.353, Z    +0.000, E1   +56.690, E3 +62146.897}
ENDSPLINE

SPLINE
SPL {X  -127.117, Y  +272.287, Z    +0.000, E1   +62.713, E3 +62316.119}
SPL {X  -152.442, Y  +313.682, Z    +0.000, E1   +51.943, E3 +62320.351}
SPL {X  -159.925, Y  +335.326, Z    +0.000, E1   +41.361, E3 +62320.293}
SPL {X  -163.450, Y  +351.595, Z    +0.000, E1   +29.785, E3 +62319.404}
SPL {X  -165.127, Y  +365.342, Z    +0.000, E1   +17.250, E3 +62319.384}
SPL {X  -165.640, Y  +376.693, Z    +0.000, E1    +4.721, E3 +62318.957}
SPL {X  -165.650, Y  +380.500, Z    +0.000, E1    -0.000, E3 +62318.108}
SPL {X  -165.650, Y  +382.123, Z    +0.000, E1    -3.912, E3 +62317.735}
SPL {X  -165.650, Y  +387.069, Z    +0.000, E1   -17.420, E3 +62317.447}
SPL {X  -165.650, Y  +393.439, Z    +0.000, E1   -35.398, E3 +62316.992}
SPL {X  -165.650, Y  +400.610, Z    +0.000, E1   -50.510, E3 +62316.730}
SPL {X  -165.650, Y  +414.376, Z    +0.000, E1   -68.098, E3 +62314.764}
SPL {X  -165.650, Y  +468.582, Z    +0.000, E1   -78.237, E3 +62323.534}
SPL {X  -158.306, Y  +724.277, Z    +0.000, E1   -77.461, E3 +62413.975}
ENDSPLINE

SPLINE
SPL {X  -160.145, Y  +717.851, Z    +0.000, E1   -75.386, E3 +62434.488}
ENDSPLINE

SPLINE
SPL {X  -157.156, Y  +727.862, Z    +0.000, E1   -75.175, E3 +62441.961}
SPL {X  -154.068, Y  +736.353, Z    +0.000, E1   -74.906, E3 +62449.135}
SPL {X  -149.738, Y  +746.340, Z    +0.000, E1   -74.451, E3 +62458.823}
SPL {X  -145.204, Y  +755.223, Z    +0.000, E1   -74.188, E3 +62465.549}
SPL {X  -142.724, Y  +759.583, Z    +0.000, E1   -73.634, E3 +62472.369}
SPL {X  -138.277, Y  +766.711, Z    +0.000, E1   -73.303, E3 +62478.499}
SPL {X  -134.662, Y  +771.969, Z    +0.000, E1   -72.884, E3 +62483.942}
SPL {X  -131.459, Y  +776.289, Z    +0.000, E1   -72.475, E3 +62488.609}
SPL {X  -128.771, Y  +779.702, Z    +0.000, E1   -71.875, E3 +62493.556}
SPL {X  -124.506, Y  +784.762, Z    +0.000, E1   -71.815, E3 +62496.444}
SPL {X  -112.958, Y  +796.663, Z    +0.000, E1   -74.119, E3 +62493.148}
SPL {X   -51.449, Y  +832.958, Z    +0.000, E1   -57.230, E3 +62652.475}
ENDSPLINE

SPLINE
SPL {X  -123.821, Y  +785.537, Z    +0.000, E1   -64.536, E3 +62854.220}
SPL {X  -153.467, Y  +737.853, Z    +0.000, E1   -51.757, E3 +62856.534}
SPL {X  -161.000, Y  +714.475, Z    +0.000, E1   -39.424, E3 +62856.007}
SPL {X  -164.534, Y  +694.695, Z    +0.000, E1   -23.511, E3 +62854.297}
SPL {X  -165.597, Y  +679.703, Z    +0.000, E1    -7.645, E3 +62854.173}
SPL {X  -165.650, Y  +673.520, Z    +0.000, E1    -0.048, E3 +62853.124}
SPL {X  -165.650, Y  +671.692, Z    +0.000, E1    +4.450, E3 +62852.691}
SPL {X  -165.650, Y  +667.743, Z    +0.000, E1   +15.617, E3 +62852.609}
SPL {X  -165.650, Y  +662.891, Z    +0.000, E1   +29.740, E3 +62852.127}
SPL {X  -165.650, Y  +655.319, Z    +0.000, E1   +47.265, E3 +62851.976}
SPL {X  -165.650, Y  +642.000, Z    +0.000, E1   +65.561, E3 +62850.957}
SPL {X  -165.650, Y  +619.979, Z    +0.000, E1   +79.465, E3 +62846.963}
SPL {X  -165.650, Y  +569.632, Z    +0.000, E1   +78.783, E3 +62862.242}
SPL {X  -158.840, Y  +331.491, Z    +0.000, E1   +77.462, E3 +62948.552}
ENDSPLINE

SPLINE
SPL {X  -159.893, Y  +335.208, Z    +0.000, E1   +75.483, E3 +62969.287}
ENDSPLINE

SPLINE
SPL {X  -156.487, Y  +324.170, Z    +0.000, E1   +75.150, E3 +62978.668}
SPL {X  -142.256, Y  +293.629, Z    +0.000, E1   +77.020, E3 +62973.768}
ENDSPLINE

SPLINE
SPL {X  -142.811, Y  +294.566, Z    +0.000, E1   +75.668, E3 +62985.730}
ENDSPLINE

SPLINE
SPL {X  -141.646, Y  +292.615, Z    +0.000, E1   +74.702, E3 +62994.824}
SPL {X  -140.419, Y  +290.622, Z    +0.000, E1   +73.705, E3 +63003.667}
SPL {X  -136.008, Y  +283.940, Z    +0.000, E1   +73.594, E3 +63007.786}
SPL {X  -132.748, Y  +279.415, Z    +0.000, E1   +73.006, E3 +63013.842}
SPL {X  -129.007, Y  +274.590, Z    +0.000, E1   +72.484, E3 +63019.191}
SPL {X  -125.914, Y  +270.864, Z    +0.000, E1   +72.144, E3 +63022.682}
SPL {X  -123.729, Y  +268.359, Z    +0.000, E1   +71.932, E3 +63024.855}
SPL {X  -111.023, Y  +255.562, Z    +0.000, E1   +75.772, E3 +63015.720}
SPL {X   -52.752, Y  +221.474, Z    +0.000, E1   +59.157, E3 +63144.972}
SPL {X   -49.901, Y  +220.545, Z    +0.000, E1   +56.696, E3 +63231.365}
ENDSPLINE

SPLINE
SPL {X  -127.117, Y  +272.287, Z    +0.000, E1   +62.713, E3 +63377.657}
SPL {X  -152.442, Y  +313.682, Z    +0.000, E1   +51.943, E3 +63381.889}
SPL {X  -162.319, Y  +345.447, Z    +0.000, E1   +34.671, E3 +63381.315}
SPL {X  -165.127, Y  +365.342, Z    +0.000, E1   +17.250, E3 +63380.923}
SPL {X  -165.640, Y  +376.693, Z    +0.000, E1    +4.721, E3 +63380.496}
SPL {X  -165.650, Y  +380.500, Z    +0.000, E1    -0.000, E3 +63379.646}
SPL {X  -165.650, Y  +383.262, Z    +0.000, E1    -6.645, E3 +63379.176}
SPL {X  -165.650, Y  +388.390, Z    +0.000, E1   -21.508, E3 +63378.963}
SPL {X  -165.650, Y  +393.439, Z    +0.000, E1   -35.398, E3 +63378.531}
SPL {X  -165.650, Y  +400.610, Z    +0.000, E1   -50.510, E3 +63378.268}
SPL {X  -165.650, Y  +414.376, Z    +0.000, E1   -68.098, E3 +63376.302}
SPL {X  -165.650, Y  +468.582, Z    +0.000, E1   -78.237, E3 +63385.072}
SPL {X  -158.306, Y  +724.277, Z    +0.000, E1   -77.461, E3 +63475.514}
ENDSPLINE

SPLINE
SPL {X  -160.145, Y  +717.851, Z    +0.000, E1   -75.386, E3 +63496.027}
ENDSPLINE

SPLINE
SPL {X  -157.156, Y  +727.862, Z    +0.000, E1   -75.175, E3 +63503.499}
SPL {X  -152.814, Y  +739.436, Z    +0.000, E1   -74.813, E3 +63513.353}
SPL {X  -147.104, Y  +751.659, Z    +0.000, E1   -74.255, E3 +63524.797}
SPL {X  -141.453, Y  +761.704, Z    +0.000, E1   -73.638, E3 +63535.010}
SPL {X  -135.914, Y  +770.196, Z    +0.000, E1   -72.974, E3 +63544.072}
SPL {X  -131.459, Y  +776.289, Z    +0.000, E1   -72.475, E3 +63550.147}
SPL {X  -128.771, Y  +779.702, Z    +0.000, E1   -71.875, E3 +63555.094}
SPL {X  -124.506, Y  +784.762, Z    +0.000, E1   -71.815, E3 +63557.982}
SPL {X  -112.958, Y  +796.663, Z    +0.000, E1   -74.119, E3 +63554.686}
SPL {X   -54.274, Y  +832.006, Z    +0.000, E1   -58.502, E3 +63686.706}
SPL {X   -50.797, Y  +833.169, Z    +0.000, E1   -57.000, E3 +63782.055}
ENDSPLINE

SPLINE
SPL {X  -113.713, Y  +795.955, Z    +0.000, E1   -65.735, E3 +63912.931}
SPL {X  -131.116, Y  +776.736, Z    +0.000, E1   -63.149, E3 +63917.462}
SPL {X  -153.467, Y  +737.853, Z    +0.000, E1   -51.757, E3 +63918.073}
SPL {X  -162.176, Y  +709.248, Z    +0.000, E1   -35.773, E3 +63917.098}
SPL {X  -164.888, Y  +691.368, Z    +0.000, E1   -20.174, E3 +63915.536}
SPL {X  -165.597, Y  +679.703, Z    +0.000, E1    -7.645, E3 +63915.711}
SPL {X  -165.650, Y  +673.520, Z    +0.000, E1    -0.048, E3 +63914.663}
SPL {X  -165.650, Y  +671.692, Z    +0.000, E1    +4.450, E3 +63914.230}
SPL {X  -165.650, Y  +667.743, Z    +0.000, E1   +15.617, E3 +63914.147}
SPL {X  -165.650, Y  +662.891, Z    +0.000, E1   +29.740, E3 +63913.665}
SPL {X  -165.650, Y  +655.319, Z    +0.000, E1   +47.265, E3 +63913.514}
SPL {X  -165.650, Y  +642.000, Z    +0.000, E1   +65.561, E3 +63912.495}
SPL {X  -165.650, Y  +619.979, Z    +0.000, E1   +79.465, E3 +63908.502}
SPL {X  -165.650, Y  +569.632, Z    +0.000, E1   +78.783, E3 +63923.781}
SPL {X  -158.840, Y  +331.491, Z    +0.000, E1   +77.462, E3 +64010.091}
ENDSPLINE

SPLINE
SPL {X  -159.893, Y  +335.208, Z    +0.000, E1   +75.483, E3 +64030.825}
ENDSPLINE

SPLINE
SPL {X  -156.487, Y  +324.170, Z    +0.000, E1   +75.150, E3 +64040.207}
SPL {X  -142.256, Y  +293.629, Z    +0.000, E1   +77.020, E3 +64035.306}
ENDSPLINE

SPLINE
SPL {X  -142.811, Y  +294.566, Z    +0.000, E1   +75.668, E3 +64047.269}
ENDSPLINE

SPLINE
SPL {X  -141.646, Y  +292.615, Z    +0.000, E1   +74.702, E3 +64056.362}
SPL {X  -140.419, Y  +290.622, Z    +0.000, E1   +73.705, E3 +64065.205}
SPL {X  -135.839, Y  +283.697, Z    +0.000, E1   +73.388, E3 +64070.944}
SPL {X  -131.336, Y  +277.551, Z    +0.000, E1   +72.879, E3 +64077.196}
SPL {X  -126.848, Y  +271.966, Z    +0.000, E1   +72.322, E3 +64082.924}
SPL {X  -123.729, Y  +268.359, Z    +0.000, E1   +71.932, E3 +64086.393}
SPL {X  -111.023, Y  +255.562, Z    +0.000, E1   +75.772, E3 +64077.259}
SPL {X   -49.289, Y  +220.353, Z    +0.000, E1   +56.690, E3 +64269.974}
ENDSPLINE

SPLINE
SPL {X  -127.117, Y  +272.287, Z    +0.000, E1   +62.713, E3 +64439.196}
SPL {X  -154.956, Y  +319.945, Z    +0.000, E1   +49.402, E3 +64443.595}
SPL {X  -162.871, Y  +348.286, Z    +0.000, E1   +32.462, E3 +64442.623}
SPL {X  -165.127, Y  +365.342, Z    +0.000, E1   +17.250, E3 +64442.461}
SPL {X  -165.640, Y  +376.693, Z    +0.000, E1    +4.721, E3 +64442.034}
SPL {X  -165.650, Y  +380.500, Z    +0.000, E1    -0.000, E3 +64441.185}
SPL {X  -165.650, Y  +383.262, Z    +0.000, E1    -6.645, E3 +64440.714}
SPL {X  -165.650, Y  +388.390, Z    +0.000, E1   -21.508, E3 +64440.502}
SPL {X  -165.650, Y  +393.439, Z    +0.000, E1   -35.398, E3 +64440.069}
SPL {X  -165.650, Y  +400.610, Z    +0.000, E1   -50.510, E3 +64439.807}
SPL {X  -165.650, Y  +414.376, Z    +0.000, E1   -68.098, E3 +64437.841}
SPL {X  -165.650, Y  +468.582, Z    +0.000, E1   -78.237, E3 +64446.611}
SPL {X  -158.306, Y  +724.277, Z    +0.000, E1   -77.461, E3 +64537.052}
ENDSPLINE

SPLINE
SPL {X  -160.145, Y  +717.851, Z    +0.000, E1   -75.386, E3 +64557.565}
ENDSPLINE

SPLINE
SPL {X  -157.156, Y  +727.862, Z    +0.000, E1   -75.175, E3 +64565.038}
SPL {X  -154.068, Y  +736.353, Z    +0.000, E1   -74.906, E3 +64572.212}
SPL {X  -149.738, Y  +746.340, Z    +0.000, E1   -74.451, E3 +64581.900}
SPL {X  -144.163, Y  +757.090, Z    +0.000, E1   -74.033, E3 +64590.992}
SPL {X  -140.473, Y  +763.291, Z    +0.000, E1   -73.478, E3 +64598.434}
SPL {X  -135.914, Y  +770.196, Z    +0.000, E1   -72.974, E3 +64605.610}
SPL {X  -131.459, Y  +776.289, Z    +0.000, E1   -72.475, E3 +64611.686}
SPL {X  -128.771, Y  +779.702, Z    +0.000, E1   -71.875, E3 +64616.632}
SPL {X  -124.506, Y  +784.762, Z    +0.000, E1   -71.815, E3 +64619.521}
SPL {X  -112.958, Y  +796.663, Z    +0.000, E1   -74.119, E3 +64616.224}
SPL {X   -51.449, Y  +832.958, Z    +0.000, E1   -57.230, E3 +64775.551}
ENDSPLINE

SPLINE
SPL {X  -123.821, Y  +785.537, Z    +0.000, E1   -64.536, E3 +64977.297}
SPL {X  -153.467, Y  +737.853, Z    +0.000, E1   -51.757, E3 +64979.611}
SPL {X  -162.176, Y  +709.248, Z    +0.000, E1   -35.773, E3 +64978.637}
SPL {X  -164.888, Y  +691.368, Z    +0.000, E1   -20.174, E3 +64977.075}
SPL {X  -165.597, Y  +679.703, Z    +0.000, E1    -7.645, E3 +64977.250}
SPL {X  -165.650, Y  +673.520, Z    +0.000, E1    -0.048, E3 +64976.201}
SPL {X  -165.650, Y  +671.692, Z    +0.000, E1    +4.450, E3 +64975.768}
SPL {X  -165.650, Y  +667.743, Z    +0.000, E1   +15.617, E3 +64975.686}
SPL {X  -165.650, Y  +661.459, Z    +0.000, E1   +33.218, E3 +64975.266}
SPL {X  -165.650, Y  +650.834, Z    +0.000, E1   +55.143, E3 +64974.654}
SPL {X  -165.650, Y  +639.785, Z    +0.000, E1   +67.512, E3 +64973.871}
SPL {X  -165.650, Y  +619.979, Z    +0.000, E1   +79.465, E3 +64970.040}
SPL {X  -165.650, Y  +569.632, Z    +0.000, E1   +78.783, E3 +64985.319}
SPL {X  -158.840, Y  +331.491, Z    +0.000, E1   +77.462, E3 +65071.629}
ENDSPLINE

SPLINE
SPL {X  -159.893, Y  +335.208, Z    +0.000, E1   +75.483, E3 +65092.364}
ENDSPLINE

SPLINE
SPL {X  -156.487, Y  +324.170, Z    +0.000, E1   +75.150, E3 +65101.745}
SPL {X  -142.256, Y  +293.629, Z    +0.000, E1   +77.020, E3 +65096.845}
ENDSPLINE

SPLINE
SPL {X  -142.811, Y  +294.566, Z    +0.000, E1   +75.668, E3 +65108.807}
ENDSPLINE

SPLINE
SPL {X  -141.646, Y  +292.615, Z    +0.000, E1   +74.702, E3 +65117.901}
SPL {X  -140.419, Y  +290.622, Z    +0.000, E1   +73.705, E3 +65126.744}
SPL {X  -136.008, Y  +283.940, Z    +0.000, E1   +73.594, E3 +65130.863}
SPL {X  -132.748, Y  +279.415, Z    +0.000, E1   +73.006, E3 +65136.919}
SPL {X  -129.007, Y  +274.590, Z    +0.000, E1   +72.484, E3 +65142.268}
SPL {X  -125.914, Y  +270.864, Z    +0.000, E1   +72.144, E3 +65145.759}
SPL {X  -123.729, Y  +268.359, Z    +0.000, E1   +71.932, E3 +65147.932}
SPL {X  -111.023, Y  +255.562, Z    +0.000, E1   +75.772, E3 +65138.797}
SPL {X   -49.289, Y  +220.353, Z    +0.000, E1   +56.690, E3 +65331.512}
ENDSPLINE

SPLINE
SPL {X  -127.117, Y  +272.287, Z    +0.000, E1   +62.713, E3 +65500.734}
SPL {X  -154.956, Y  +319.945, Z    +0.000, E1   +49.402, E3 +65505.133}
SPL {X  -162.871, Y  +348.286, Z    +0.000, E1   +32.462, E3 +65504.161}
SPL {X  -165.127, Y  +365.342, Z    +0.000, E1   +17.250, E3 +65504.000}
SPL {X  -165.640, Y  +376.693, Z    +0.000, E1    +4.721, E3 +65503.572}
SPL {X  -165.650, Y  +380.500, Z    +0.000, E1    -0.000, E3 +65502.723}
SPL {X  -165.650, Y  +383.262, Z    +0.000, E1    -6.645, E3 +65502.253}
SPL {X  -165.650, Y  +388.390, Z    +0.000, E1   -21.508, E3 +65502.040}
SPL {X  -165.650, Y  +393.439, Z    +0.000, E1   -35.398, E3 +65501.608}
SPL {X  -165.650, Y  +400.610, Z    +0.000, E1   -50.510, E3 +65501.345}
SPL {X  -165.650, Y  +414.376, Z    +0.000, E1   -68.098, E3 +65499.379}
SPL {X  -165.650, Y  +468.582, Z    +0.000, E1   -78.237, E3 +65508.149}
SPL {X  -158.306, Y  +724.277, Z    +0.000, E1   -77.461, E3 +65598.591}
ENDSPLINE

SPLINE
SPL {X  -160.145, Y  +717.851, Z    +0.000, E1   -75.386, E3 +65619.104}
ENDSPLINE

SPLINE
SPL {X  -157.156, Y  +727.862, Z    +0.000, E1   -75.175, E3 +65626.576}
SPL {X  -154.068, Y  +736.353, Z    +0.000, E1   -74.906, E3 +65633.751}
SPL {X  -149.738, Y  +746.340, Z    +0.000, E1   -74.451, E3 +65643.438}
SPL {X  -144.163, Y  +757.090, Z    +0.000, E1   -74.033, E3 +65652.531}
SPL {X  -140.473, Y  +763.291, Z    +0.000, E1   -73.478, E3 +65659.972}
SPL {X  -135.914, Y  +770.196, Z    +0.000, E1   -72.974, E3 +65667.148}
SPL {X  -131.459, Y  +776.289, Z    +0.000, E1   -72.475, E3 +65673.224}
SPL {X  -128.771, Y  +779.702, Z    +0.000, E1   -71.875, E3 +65678.171}
SPL {X  -124.506, Y  +784.762, Z    +0.000, E1   -71.815, E3 +65681.059}
SPL {X  -112.958, Y  +796.663, Z    +0.000, E1   -74.119, E3 +65677.763}
SPL {X   -51.449, Y  +832.958, Z    +0.000, E1   -57.230, E3 +65837.090}
ENDSPLINE

SPLINE
SPL {X  -123.821, Y  +785.537, Z    +0.000, E1   -64.536, E3 +66038.835}
SPL {X  -153.467, Y  +737.853, Z    +0.000, E1   -51.757, E3 +66041.150}
SPL {X  -162.176, Y  +709.248, Z    +0.000, E1   -35.773, E3 +66040.175}
SPL {X  -164.888, Y  +691.368, Z    +0.000, E1   -20.174, E3 +66038.613}
SPL {X  -165.597, Y  +679.703, Z    +0.000, E1    -7.645, E3 +66038.788}
SPL {X  -165.650, Y  +673.520, Z    +0.000, E1    -0.048, E3 +66037.740}
SPL {X  -165.650, Y  +671.692, Z    +0.000, E1    +4.450, E3 +66037.306}
SPL {X  -165.650, Y  +667.743, Z    +0.000, E1   +15.617, E3 +66037.224}
SPL {X  -165.650, Y  +661.459, Z    +0.000, E1   +33.218, E3 +66036.805}
SPL {X  -165.650, Y  +650.834, Z    +0.000, E1   +55.143, E3 +66036.193}
SPL {X  -165.650, Y  +639.785, Z    +0.000, E1   +67.512, E3 +66035.410}
SPL {X  -165.650, Y  +619.979, Z    +0.000, E1   +79.465, E3 +66031.579}
SPL {X  -165.650, Y  +569.632, Z    +0.000, E1   +78.783, E3 +66046.858}
SPL {X  -158.840, Y  +331.491, Z    +0.000, E1   +77.462, E3 +66133.168}
ENDSPLINE

SPLINE
SPL {X  -159.893, Y  +335.208, Z    +0.000, E1   +75.483, E3 +66153.902}
ENDSPLINE

SPLINE
SPL {X  -156.487, Y  +324.170, Z    +0.000, E1   +75.150, E3 +66163.283}
SPL {X  -142.256, Y  +293.629, Z    +0.000, E1   +77.020, E3 +66158.383}
ENDSPLINE

SPLINE
SPL {X  -142.811, Y  +294.566, Z    +0.000, E1   +75.668, E3 +66170.346}
ENDSPLINE

SPLINE
SPL {X  -141.646, Y  +292.615, Z    +0.000, E1   +74.702, E3 +66179.439}
SPL {X  -140.419, Y  +290.622, Z    +0.000, E1   +73.705, E3 +66188.282}
SPL {X  -136.008, Y  +283.940, Z    +0.000, E1   +73.594, E3 +66192.401}
SPL {X  -132.748, Y  +279.415, Z    +0.000, E1   +73.006, E3 +66198.457}
SPL {X  -129.007, Y  +274.590, Z    +0.000, E1   +72.484, E3 +66203.806}
SPL {X  -125.914, Y  +270.864, Z    +0.000, E1   +72.144, E3 +66207.298}
SPL {X  -123.729, Y  +268.359, Z    +0.000, E1   +71.932, E3 +66209.470}
SPL {X  -111.023, Y  +255.562, Z    +0.000, E1   +75.772, E3 +66200.336}
SPL {X   -49.289, Y  +220.353, Z    +0.000, E1   +56.690, E3 +66393.051}
ENDSPLINE

SPLINE
SPL {X  -127.117, Y  +272.287, Z    +0.000, E1   +62.713, E3 +66562.273}
SPL {X  -154.956, Y  +319.945, Z    +0.000, E1   +49.402, E3 +66566.672}
SPL {X  -162.871, Y  +348.286, Z    +0.000, E1   +32.462, E3 +66565.699}
SPL {X  -165.127, Y  +365.342, Z    +0.000, E1   +17.250, E3 +66565.538}
SPL {X  -165.640, Y  +376.693, Z    +0.000, E1    +4.721, E3 +66565.111}
SPL {X  -165.650, Y  +380.500, Z    +0.000, E1    -0.000, E3 +66564.262}
SPL {X  -165.650, Y  +383.262, Z    +0.000, E1    -6.645, E3 +66563.791}
SPL {X  -165.650, Y  +388.390, Z    +0.000, E1   -21.508, E3 +66563.579}
SPL {X  -165.650, Y  +393.439, Z    +0.000, E1   -35.398, E3 +66563.146}
SPL {X  -165.650, Y  +400.610, Z    +0.000, E1   -50.510, E3 +66562.884}
SPL {X  -165.650, Y  +414.376, Z    +0.000, E1   -68.098, E3 +66560.917}
SPL {X  -165.650, Y  +468.582, Z    +0.000, E1   -78.237, E3 +66569.688}
SPL {X  -158.306, Y  +724.277, Z    +0.000, E1   -77.461, E3 +66660.129}
ENDSPLINE

SPLINE
SPL {X  -160.145, Y  +717.851, Z    +0.000, E1   -75.386, E3 +66680.642}
ENDSPLINE

SPLINE
SPL {X  -157.156, Y  +727.862, Z    +0.000, E1   -75.175, E3 +66688.114}
SPL {X  -154.068, Y  +736.353, Z    +0.000, E1   -74.906, E3 +66695.289}
SPL {X  -149.738, Y  +746.340, Z    +0.000, E1   -74.451, E3 +66704.977}
SPL {X  -144.163, Y  +757.090, Z    +0.000, E1   -74.033, E3 +66714.069}
SPL {X  -140.473, Y  +763.291, Z    +0.000, E1   -73.478, E3 +66721.511}
SPL {X  -135.914, Y  +770.196, Z    +0.000, E1   -72.974, E3 +66728.687}
SPL {X  -131.459, Y  +776.289, Z    +0.000, E1   -72.475, E3 +66734.763}
SPL {X  -128.771, Y  +779.702, Z    +0.000, E1   -71.875, E3 +66739.709}
SPL {X  -124.506, Y  +784.762, Z    +0.000, E1   -71.815, E3 +66742.598}
SPL {X  -112.958, Y  +796.663, Z    +0.000, E1   -74.119, E3 +66739.301}
SPL {X   -51.449, Y  +832.958, Z    +0.000, E1   -57.230, E3 +66898.628}
ENDSPLINE

SPLINE
SPL {X  -123.821, Y  +785.537, Z    +0.000, E1   -64.536, E3 +67100.374}
SPL {X  -153.467, Y  +737.853, Z    +0.000, E1   -51.757, E3 +67102.688}
SPL {X  -162.176, Y  +709.248, Z    +0.000, E1   -35.773, E3 +67101.714}
SPL {X  -164.888, Y  +691.368, Z    +0.000, E1   -20.174, E3 +67100.151}
SPL {X  -165.597, Y  +679.703, Z    +0.000, E1    -7.645, E3 +67100.327}
SPL {X  -165.650, Y  +673.520, Z    +0.000, E1    -0.048, E3 +67099.278}
SPL {X  -165.650, Y  +671.692, Z    +0.000, E1    +4.450, E3 +67098.845}
SPL {X  -165.650, Y  +667.743, Z    +0.000, E1   +15.617, E3 +67098.763}
SPL {X  -165.650, Y  +661.459, Z    +0.000, E1   +33.218, E3 +67098.343}
SPL {X  -165.650, Y  +650.834, Z    +0.000, E1   +55.143, E3 +67097.731}
SPL {X  -165.650, Y  +639.785, Z    +0.000, E1   +67.512, E3 +67096.948}
SPL {X  -165.650, Y  +619.979, Z    +0.000, E1   +79.465, E3 +67093.117}
SPL {X  -165.650, Y  +569.632, Z    +0.000, E1   +78.783, E3 +67108.396}
SPL {X  -158.840, Y  +331.491, Z    +0.000, E1   +77.462, E3 +67194.706}
ENDSPLINE

SPLINE
SPL {X  -159.893, Y  +335.208, Z    +0.000, E1   +75.483, E3 +67215.441}
ENDSPLINE

SPLINE
SPL {X  -156.487, Y  +324.170, Z    +0.000, E1   +75.150, E3 +67224.822}
SPL {X  -142.256, Y  +293.629, Z    +0.000, E1   +77.020, E3 +67219.922}
ENDSPLINE

SPLINE
SPL {X  -142.811, Y  +294.566, Z    +0.000, E1   +75.668, E3 +67231.884}
ENDSPLINE

SPLINE
SPL {X  -141.646, Y  +292.615, Z    +0.000, E1   +74.702, E3 +67240.978}
SPL {X  -140.419, Y  +290.622, Z    +0.000, E1   +73.705, E3 +67249.821}
SPL {X  -136.008, Y  +283.940, Z    +0.000, E1   +73.594, E3 +67253.940}
SPL {X  -132.748, Y  +279.415, Z    +0.000, E1   +73.006, E3 +67259.996}
SPL {X  -129.007, Y  +274.590, Z    +0.000, E1   +72.484, E3 +67265.345}
SPL {X  -125.914, Y  +270.864, Z    +0.000, E1   +72.144, E3 +67268.836}
SPL {X  -123.729, Y  +268.359, Z    +0.000, E1   +71.932, E3 +67271.008}
SPL {X  -111.023, Y  +255.562, Z    +0.000, E1   +75.772, E3 +67261.874}
SPL {X   -49.289, Y  +220.353, Z    +0.000, E1   +56.690, E3 +67454.589}
ENDSPLINE

SPLINE
SPL {X  -127.117, Y  +272.287, Z    +0.000, E1   +62.713, E3 +67623.811}
SPL {X  -154.956, Y  +319.945, Z    +0.000, E1   +49.402, E3 +67628.210}
SPL {X  -162.871, Y  +348.286, Z    +0.000, E1   +32.462, E3 +67627.238}
SPL {X  -165.127, Y  +365.342, Z    +0.000, E1   +17.250, E3 +67627.076}
SPL {X  -165.640, Y  +376.693, Z    +0.000, E1    +4.721, E3 +67626.649}
SPL {X  -165.650, Y  +380.500, Z    +0.000, E1    -0.000, E3 +67625.800}
SPL {X  -165.650, Y  +383.262, Z    +0.000, E1    -6.645, E3 +67625.329}
SPL {X  -165.650, Y  +388.390, Z    +0.000, E1   -21.508, E3 +67625.117}
SPL {X  -165.650, Y  +393.439, Z    +0.000, E1   -35.398, E3 +67624.685}
SPL {X  -165.650, Y  +400.610, Z    +0.000, E1   -50.510, E3 +67624.422}
SPL {X  -165.650, Y  +414.376, Z    +0.000, E1   -68.098, E3 +67622.456}
SPL {X  -165.650, Y  +468.582, Z    +0.000, E1   -78.237, E3 +67631.226}
SPL {X  -158.306, Y  +724.277, Z    +0.000, E1   -77.461, E3 +67721.667}
ENDSPLINE

SPLINE
SPL {X  -160.145, Y  +717.851, Z    +0.000, E1   -75.386, E3 +67742.181}
ENDSPLINE

SPLINE
SPL {X  -157.156, Y  +727.862, Z    +0.000, E1   -75.175, E3 +67749.653}
SPL {X  -152.814, Y  +739.436, Z    +0.000, E1   -74.813, E3 +67759.507}
SPL {X  -147.104, Y  +751.659, Z    +0.000, E1   -74.255, E3 +67770.951}
SPL {X  -141.453, Y  +761.704, Z    +0.000, E1   -73.638, E3 +67781.164}
SPL {X  -135.914, Y  +770.196, Z    +0.000, E1   -72.974, E3 +67790.225}
SPL {X  -131.459, Y  +776.289, Z    +0.000, E1   -72.475, E3 +67796.301}
SPL {X  -127.605, Y  +781.126, Z    +0.000, E1   -71.922, E3 +67801.745}
SPL {X  -124.773, Y  +784.457, Z    +0.000, E1   -71.383, E3 +67805.793}
SPL {X  -119.086, Y  +790.645, Z    +0.000, E1   -72.931, E3 +67802.647}
SPL {X   -51.449, Y  +832.958, Z    +0.000, E1   -57.230, E3 +67960.167}
ENDSPLINE

SPLINE
SPL {X  -123.821, Y  +785.537, Z    +0.000, E1   -64.536, E3 +68161.912}
SPL {X  -153.467, Y  +737.853, Z    +0.000, E1   -51.757, E3 +68164.227}
SPL {X  -162.176, Y  +709.248, Z    +0.000, E1   -35.773, E3 +68163.252}
SPL {X  -164.888, Y  +691.368, Z    +0.000, E1   -20.174, E3 +68161.690}
SPL {X  -165.597, Y  +679.703, Z    +0.000, E1    -7.645, E3 +68161.865}
SPL {X  -165.650, Y  +673.520, Z    +0.000, E1    -0.048, E3 +68160.817}
SPL {X  -165.650, Y  +671.692, Z    +0.000, E1    +4.450, E3 +68160.383}
SPL {X  -165.650, Y  +667.743, Z    +0.000, E1   +15.617, E3 +68160.301}
SPL {X  -165.650, Y  +661.459, Z    +0.000, E1   +33.218, E3 +68159.882}
SPL {X  -165.650, Y  +653.296, Z    +0.000, E1   +51.333, E3 +68159.437}
SPL {X  -165.650, Y  +642.000, Z    +0.000, E1   +65.561, E3 +68158.649}
SPL {X  -165.650, Y  +619.979, Z    +0.000, E1   +79.465, E3 +68154.656}
SPL {X  -165.650, Y  +584.722, Z    +0.000, E1   +79.551, E3 +68163.947}
SPL {X  -165.650, Y  +560.326, Z    +0.000, E1   +78.360, E3 +68173.669}
SPL {X  -160.258, Y  +336.579, Z    +0.000, E1   +78.314, E3 +68245.191}
SPL {X  -159.618, Y  +334.207, Z    +0.000, E1   +75.622, E3 +68276.005}
SPL {X  -157.855, Y  +328.284, Z    +0.000, E1   +75.167, E3 +68283.970}
SPL {X  -155.139, Y  +320.432, Z    +0.000, E1   +75.106, E3 +68288.647}
SPL {X  -142.256, Y  +293.629, Z    +0.000, E1   +77.020, E3 +68281.460}
ENDSPLINE

SPLINE
SPL {X  -142.811, Y  +294.566, Z    +0.000, E1   +75.668, E3 +68293.422}
ENDSPLINE

SPLINE
SPL {X  -141.646, Y  +292.615, Z    +0.000, E1   +74.702, E3 +68302.516}
SPL {X  -140.419, Y  +290.622, Z    +0.000, E1   +73.705, E3 +68311.359}
SPL {X  -136.008, Y  +283.940, Z    +0.000, E1   +73.594, E3 +68315.478}
SPL {X  -131.988, Y  +278.404, Z    +0.000, E1   +72.860, E3 +68323.033}
SPL {X  -126.848, Y  +271.966, Z    +0.000, E1   +72.322, E3 +68329.078}
SPL {X  -123.729, Y  +268.359, Z    +0.000, E1   +71.932, E3 +68332.547}
SPL {X  -111.023, Y  +255.562, Z    +0.000, E1   +75.772, E3 +68323.413}
SPL {X   -49.289, Y  +220.353, Z    +0.000, E1   +56.690, E3 +68516.128}
ENDSPLINE

SPLINE
SPL {X  -127.117, Y  +272.287, Z    +0.000, E1   +62.713, E3 +68685.350}
SPL {X  -152.442, Y  +313.682, Z    +0.000, E1   +51.943, E3 +68689.581}
SPL {X  -159.925, Y  +335.326, Z    +0.000, E1   +41.361, E3 +68689.523}
SPL {X  -163.450, Y  +351.595, Z    +0.000, E1   +29.785, E3 +68688.635}
SPL {X  -165.127, Y  +365.342, Z    +0.000, E1   +17.250, E3 +68688.615}
SPL {X  -165.640, Y  +376.693, Z    +0.000, E1    +4.721, E3 +68688.188}
SPL {X  -165.650, Y  +380.500, Z    +0.000, E1    -0.000, E3 +68687.339}
SPL {X  -165.650, Y  +382.123, Z    +0.000, E1    -3.912, E3 +68686.966}
SPL {X  -165.650, Y  +387.069, Z    +0.000, E1   -17.420, E3 +68686.677}
SPL {X  -165.650, Y  +393.439, Z    +0.000, E1   -35.398, E3 +68686.223}
SPL {X  -165.650, Y  +400.610, Z    +0.000, E1   -50.510, E3 +68685.961}
SPL {X  -165.650, Y  +414.376, Z    +0.000, E1   -68.098, E3 +68683.994}
SPL {X  -165.650, Y  +468.582, Z    +0.000, E1   -78.237, E3 +68692.765}
SPL {X  -160.244, Y  +717.475, Z    +0.000, E1   -78.917, E3 +68765.322}
SPL {X  -159.651, Y  +719.676, Z    +0.000, E1   -75.661, E3 +68801.709}
SPL {X  -157.156, Y  +727.862, Z    +0.000, E1   -75.175, E3 +68811.191}
SPL {X  -152.814, Y  +739.436, Z    +0.000, E1   -74.813, E3 +68821.045}
SPL {X  -148.754, Y  +748.385, Z    +0.000, E1   -74.281, E3 +68830.487}
SPL {X  -144.163, Y  +757.090, Z    +0.000, E1   -74.033, E3 +68837.146}
SPL {X  -140.473, Y  +763.291, Z    +0.000, E1   -73.478, E3 +68844.588}
SPL {X  -135.914, Y  +770.196, Z    +0.000, E1   -72.974, E3 +68851.764}
SPL {X  -131.459, Y  +776.289, Z    +0.000, E1   -72.475, E3 +68857.840}
SPL {X  -128.771, Y  +779.702, Z    +0.000, E1   -71.875, E3 +68862.786}
SPL {X  -125.267, Y  +783.889, Z    +0.000, E1   -71.674, E3 +68865.899}
SPL {X  -119.086, Y  +790.645, Z    +0.000, E1   -72.931, E3 +68864.185}
SPL {X   -51.449, Y  +832.958, Z    +0.000, E1   -57.230, E3 +69021.705}
ENDSPLINE

SPLINE
SPL {X  -123.821, Y  +785.537, Z    +0.000, E1   -64.536, E3 +69223.450}
SPL {X  -153.467, Y  +737.853, Z    +0.000, E1   -51.757, E3 +69225.765}
SPL {X  -161.000, Y  +714.475, Z    +0.000, E1   -39.424, E3 +69225.238}
SPL {X  -164.534, Y  +694.695, Z    +0.000, E1   -23.511, E3 +69223.528}
SPL {X  -165.597, Y  +679.703, Z    +0.000, E1    -7.645, E3 +69223.403}
SPL {X  -165.650, Y  +673.520, Z    +0.000, E1    -0.048, E3 +69222.355}
SPL {X  -165.650, Y  +671.692, Z    +0.000, E1    +4.450, E3 +69221.922}
SPL {X  -165.650, Y  +667.743, Z    +0.000, E1   +15.617, E3 +69221.840}
SPL {X  -165.650, Y  +662.891, Z    +0.000, E1   +29.740, E3 +69221.358}
SPL {X  -165.650, Y  +655.319, Z    +0.000, E1   +47.265, E3 +69221.206}
SPL {X  -165.650, Y  +642.000, Z    +0.000, E1   +65.561, E3 +69220.188}
SPL {X  -165.650, Y  +619.979, Z    +0.000, E1   +79.465, E3 +69216.194}
SPL {X  -165.650, Y  +569.632, Z    +0.000, E1   +78.783, E3 +69231.473}
SPL {X  -158.840, Y  +331.491, Z    +0.000, E1   +77.462, E3 +69317.783}
ENDSPLINE

SPLINE
SPL {X  -159.893, Y  +335.208, Z    +0.000, E1   +75.483, E3 +69338.518}
ENDSPLINE

SPLINE
SPL {X  -156.487, Y  +324.170, Z    +0.000, E1   +75.150, E3 +69347.899}
SPL {X  -142.256, Y  +293.629, Z    +0.000, E1   +77.020, E3 +69342.999}
ENDSPLINE

SPLINE
SPL {X  -142.811, Y  +294.566, Z    +0.000, E1   +75.668, E3 +69354.961}
ENDSPLINE

SPLINE
SPL {X  -142.084, Y  +293.340, Z    +0.000, E1   +74.562, E3 +69364.923}
ENDSPLINE

SPLINE
SPL {X  -144.490, Y  +297.490, Z    +0.000, E1   +72.455, E3 +69379.480}
ENDSPLINE

SPLINE
SPL {X  -140.483, Y  +290.724, Z    +0.000, E1   +71.922, E3 +69387.156}
SPL {X  -136.362, Y  +284.451, Z    +0.000, E1   +71.514, E3 +69393.322}
SPL {X  -132.604, Y  +279.221, Z    +0.000, E1   +70.988, E3 +69399.351}
SPL {X  -129.663, Y  +275.410, Z    +0.000, E1   +70.632, E3 +69403.275}
SPL {X  -127.149, Y  +272.325, Z    +0.000, E1   +70.073, E3 +69407.655}
SPL {X  -123.924, Y  +268.578, Z    +0.000, E1   +70.633, E3 +69407.471}
SPL {X  -115.163, Y  +259.431, Z    +0.000, E1   +74.058, E3 +69398.581}
SPL {X   -55.479, Y  +222.417, Z    +0.000, E1   +56.403, E3 +69584.435}
ENDSPLINE

SPLINE
SPL {X  -130.757, Y  +276.802, Z    +0.000, E1   +58.343, E3 +69740.371}
SPL {X  -154.788, Y  +319.502, Z    +0.000, E1   +45.389, E3 +69744.569}
SPL {X  -161.887, Y  +343.393, Z    +0.000, E1   +32.461, E3 +69745.026}
SPL {X  -164.949, Y  +363.277, Z    +0.000, E1   +17.059, E3 +69744.300}
SPL {X  -165.638, Y  +376.493, Z    +0.000, E1    +4.395, E3 +69743.939}
SPL {X  -165.650, Y  +380.500, Z    +0.000, E1    +0.000, E3 +69743.049}
SPL {X  -165.650, Y  +381.832, Z    +0.000, E1    -2.686, E3 +69742.521}
SPL {X  -165.650, Y  +385.053, Z    +0.000, E1   -10.073, E3 +69742.427}
SPL {X  -165.650, Y  +388.847, Z    +0.000, E1   -19.524, E3 +69742.391}
SPL {X  -165.650, Y  +393.562, Z    +0.000, E1   -31.212, E3 +69741.875}
SPL {X  -165.650, Y  +400.090, Z    +0.000, E1   -44.561, E3 +69741.729}
SPL {X  -165.650, Y  +415.429, Z    +0.000, E1   -64.815, E3 +69739.788}
SPL {X  -165.650, Y  +470.008, Z    +0.000, E1   -77.011, E3 +69748.332}
SPL {X  -160.882, Y  +714.957, Z    +0.000, E1   -77.470, E3 +69832.038}
ENDSPLINE

SPLINE
SPL {X  -163.522, Y  +701.969, Z    +0.000, E1   -74.236, E3 +69861.694}
ENDSPLINE

SPLINE
SPL {X  -160.284, Y  +717.322, Z    +0.000, E1   -73.988, E3 +69873.027}
SPL {X  -156.453, Y  +729.928, Z    +0.000, E1   -73.507, E3 +69885.179}
SPL {X  -152.193, Y  +740.900, Z    +0.000, E1   -73.135, E3 +69894.745}
SPL {X  -148.880, Y  +748.126, Z    +0.000, E1   -72.716, E3 +69902.526}
SPL {X  -144.434, Y  +756.610, Z    +0.000, E1   -72.338, E3 +69910.376}
SPL {X  -141.532, Y  +761.573, Z    +0.000, E1   -71.800, E3 +69917.017}
SPL {X  -138.580, Y  +766.249, Z    +0.000, E1   -71.449, E3 +69922.078}
SPL {X  -134.851, Y  +771.704, Z    +0.000, E1   -71.081, E3 +69927.473}
SPL {X  -131.668, Y  +776.015, Z    +0.000, E1   -70.566, E3 +69932.747}
SPL {X  -128.114, Y  +780.508, Z    +0.000, E1   -70.155, E3 +69937.342}
SPL {X  -123.825, Y  +785.533, Z    +0.000, E1   -70.642, E3 +69938.091}
SPL {X  -111.068, Y  +798.397, Z    +0.000, E1   -72.944, E3 +69935.535}
SPL {X   -54.135, Y  +832.054, Z    +0.000, E1   -56.519, E3 +70111.554}
ENDSPLINE

SPLINE
SPL {X  -119.915, Y  +789.781, Z    +0.000, E1   -62.637, E3 +70279.169}
SPL {X  -140.675, Y  +762.967, Z    +0.000, E1   -56.489, E3 +70279.511}
SPL {X  -155.138, Y  +733.569, Z    +0.000, E1   -46.550, E3 +70281.816}
SPL {X  -161.585, Y  +711.971, Z    +0.000, E1   -34.503, E3 +70280.866}
SPL {X  -164.796, Y  +692.295, Z    +0.000, E1   -19.289, E3 +70280.901}
SPL {X  -165.632, Y  +677.938, Z    +0.000, E1    -5.073, E3 +70280.272}
SPL {X  -165.650, Y  +673.500, Z    +0.000, E1    +0.000, E3 +70279.306}
SPL {X  -165.650, Y  +671.349, Z    +0.000, E1    +4.619, E3 +70278.810}
SPL {X  -165.650, Y  +666.568, Z    +0.000, E1   +16.799, E3 +70278.686}
SPL {X  -165.650, Y  +661.246, Z    +0.000, E1   +30.569, E3 +70278.466}
SPL {X  -165.650, Y  +652.403, Z    +0.000, E1   +48.665, E3 +70278.104}
SPL {X  -165.650, Y  +637.100, Z    +0.000, E1   +69.106, E3 +70274.444}
SPL {X  -165.650, Y  +616.344, Z    +0.000, E1   +74.941, E3 +70277.694}
SPL {X  -165.650, Y  +575.817, Z    +0.000, E1   +77.800, E3 +70286.623}
SPL {X  -162.613, Y  +346.923, Z    +0.000, E1   +78.263, E3 +70358.296}
SPL {X  -161.207, Y  +340.393, Z    +0.000, E1   +75.705, E3 +70388.159}
SPL {X  -146.302, Y  +300.811, Z    +0.000, E1   +78.008, E3 +70379.040}
ENDSPLINE

SPLINE
SPL {X  -147.825, Y  +303.750, Z    +0.000, E1   +76.548, E3 +70393.472}
SPL {X  -148.167, Y  +304.430, Z    +0.000, E1   +75.276, E3 +70405.565}
ENDSPLINE

SPLINE
SPL {X  -146.983, Y  +302.107, Z    +0.000, E1   +74.473, E3 +70414.046}
SPL {X  -146.624, Y  +301.420, Z    +0.000, E1   +73.294, E3 +70424.529}
SPL {X  -144.830, Y  +298.101, Z    +0.000, E1   +72.333, E3 +70434.053}
SPL {X  -140.483, Y  +290.724, Z    +0.000, E1   +71.922, E3 +70441.210}
SPL {X  -136.362, Y  +284.451, Z    +0.000, E1   +71.514, E3 +70447.376}
SPL {X  -133.329, Y  +280.198, Z    +0.000, E1   +71.389, E3 +70450.461}
SPL {X  -130.835, Y  +276.902, Z    +0.000, E1   +70.642, E3 +70456.458}
SPL {X  -127.149, Y  +272.325, Z    +0.000, E1   +70.073, E3 +70461.709}
SPL {X  -123.924, Y  +268.578, Z    +0.000, E1   +70.633, E3 +70461.525}
SPL {X  -115.163, Y  +259.431, Z    +0.000, E1   +74.058, E3 +70452.635}
SPL {X   -55.479, Y  +222.417, Z    +0.000, E1   +56.403, E3 +70638.489}
ENDSPLINE

SPLINE
SPL {X  -130.757, Y  +276.802, Z    +0.000, E1   +58.343, E3 +70794.425}
SPL {X  -154.788, Y  +319.502, Z    +0.000, E1   +45.389, E3 +70798.624}
SPL {X  -161.887, Y  +343.393, Z    +0.000, E1   +32.461, E3 +70799.080}
SPL {X  -164.949, Y  +363.277, Z    +0.000, E1   +17.059, E3 +70798.354}
SPL {X  -165.638, Y  +376.493, Z    +0.000, E1    +4.395, E3 +70797.993}
SPL {X  -165.650, Y  +380.500, Z    +0.000, E1    +0.000, E3 +70797.103}
SPL {X  -165.650, Y  +381.832, Z    +0.000, E1    -2.686, E3 +70796.575}
SPL {X  -165.650, Y  +385.053, Z    +0.000, E1   -10.073, E3 +70796.481}
SPL {X  -165.650, Y  +388.847, Z    +0.000, E1   -19.524, E3 +70796.445}
SPL {X  -165.650, Y  +393.562, Z    +0.000, E1   -31.212, E3 +70795.929}
SPL {X  -165.650, Y  +400.090, Z    +0.000, E1   -44.561, E3 +70795.783}
SPL {X  -165.650, Y  +412.079, Z    +0.000, E1   -62.360, E3 +70793.682}
SPL {X  -165.650, Y  +422.274, Z    +0.000, E1   -68.953, E3 +70794.169}
SPL {X  -165.650, Y  +460.635, Z    +0.000, E1   -76.744, E3 +70799.739}
SPL {X  -165.650, Y  +476.745, Z    +0.000, E1   -77.150, E3 +70804.291}
SPL {X  -161.095, Y  +714.078, Z    +0.000, E1   -78.221, E3 +70877.921}
ENDSPLINE

SPLINE
SPL {X  -163.418, Y  +702.603, Z    +0.000, E1   -74.313, E3 +70915.317}
ENDSPLINE

SPLINE
SPL {X  -160.284, Y  +717.322, Z    +0.000, E1   -73.988, E3 +70927.081}
SPL {X  -156.453, Y  +729.928, Z    +0.000, E1   -73.507, E3 +70939.233}
SPL {X  -152.193, Y  +740.900, Z    +0.000, E1   -73.135, E3 +70948.799}
SPL {X  -148.880, Y  +748.126, Z    +0.000, E1   -72.716, E3 +70956.581}
SPL {X  -145.823, Y  +754.085, Z    +0.000, E1   -72.288, E3 +70963.352}
SPL {X  -141.906, Y  +760.955, Z    +0.000, E1   -72.057, E3 +70969.043}
SPL {X  -138.580, Y  +766.249, Z    +0.000, E1   -71.449, E3 +70976.132}
SPL {X  -134.851, Y  +771.704, Z    +0.000, E1   -71.081, E3 +70981.528}
SPL {X  -131.668, Y  +776.015, Z    +0.000, E1   -70.566, E3 +70986.801}
SPL {X  -128.114, Y  +780.508, Z    +0.000, E1   -70.155, E3 +70991.397}
SPL {X  -123.825, Y  +785.533, Z    +0.000, E1   -70.642, E3 +70992.145}
SPL {X  -111.068, Y  +798.397, Z    +0.000, E1   -72.944, E3 +70989.589}
SPL {X   -54.135, Y  +832.054, Z    +0.000, E1   -56.519, E3 +71165.608}
ENDSPLINE

SPLINE
SPL {X  -119.915, Y  +789.781, Z    +0.000, E1   -62.637, E3 +71333.223}
SPL {X  -140.675, Y  +762.967, Z    +0.000, E1   -56.489, E3 +71333.565}
SPL {X  -155.138, Y  +733.569, Z    +0.000, E1   -46.550, E3 +71335.870}
SPL {X  -161.585, Y  +711.971, Z    +0.000, E1   -34.503, E3 +71334.920}
SPL {X  -164.796, Y  +692.295, Z    +0.000, E1   -19.289, E3 +71334.955}
SPL {X  -165.632, Y  +677.938, Z    +0.000, E1    -5.073, E3 +71334.326}
SPL {X  -165.650, Y  +673.500, Z    +0.000, E1    +0.000, E3 +71333.360}
SPL {X  -165.650, Y  +671.349, Z    +0.000, E1    +4.619, E3 +71332.864}
SPL {X  -165.650, Y  +666.568, Z    +0.000, E1   +16.799, E3 +71332.740}
SPL {X  -165.650, Y  +661.246, Z    +0.000, E1   +30.569, E3 +71332.520}
SPL {X  -165.650, Y  +652.403, Z    +0.000, E1   +48.665, E3 +71332.158}
SPL {X  -165.650, Y  +637.100, Z    +0.000, E1   +69.106, E3 +71328.498}
SPL {X  -165.650, Y  +616.344, Z    +0.000, E1   +74.941, E3 +71331.748}
SPL {X  -165.650, Y  +575.817, Z    +0.000, E1   +77.800, E3 +71340.677}
SPL {X  -161.405, Y  +341.238, Z    +0.000, E1   +76.606, E3 +71431.977}
SPL {X  -146.302, Y  +300.811, Z    +0.000, E1   +78.008, E3 +71433.094}
ENDSPLINE

SPLINE
SPL {X  -147.825, Y  +303.750, Z    +0.000, E1   +76.548, E3 +71447.526}
SPL {X  -148.167, Y  +304.430, Z    +0.000, E1   +75.276, E3 +71459.619}
ENDSPLINE

SPLINE
SPL {X  -146.983, Y  +302.107, Z    +0.000, E1   +74.473, E3 +71468.100}
SPL {X  -146.624, Y  +301.420, Z    +0.000, E1   +73.294, E3 +71478.583}
SPL {X  -144.830, Y  +298.101, Z    +0.000, E1   +72.333, E3 +71488.107}
SPL {X  -140.483, Y  +290.724, Z    +0.000, E1   +71.922, E3 +71495.264}
SPL {X  -136.362, Y  +284.451, Z    +0.000, E1   +71.514, E3 +71501.431}
SPL {X  -132.604, Y  +279.221, Z    +0.000, E1   +70.988, E3 +71507.459}
SPL {X  -129.663, Y  +275.410, Z    +0.000, E1   +70.632, E3 +71511.383}
SPL {X  -127.149, Y  +272.325, Z    +0.000, E1   +70.073, E3 +71515.763}
SPL {X  -123.924, Y  +268.578, Z    +0.000, E1   +70.633, E3 +71515.579}
SPL {X  -115.163, Y  +259.431, Z    +0.000, E1   +74.058, E3 +71506.689}
SPL {X   -55.479, Y  +222.417, Z    +0.000, E1   +56.403, E3 +71692.543}
ENDSPLINE

SPLINE
SPL {X  -130.757, Y  +276.802, Z    +0.000, E1   +58.343, E3 +71848.479}
SPL {X  -154.788, Y  +319.502, Z    +0.000, E1   +45.389, E3 +71852.678}
SPL {X  -161.887, Y  +343.393, Z    +0.000, E1   +32.461, E3 +71853.134}
SPL {X  -164.949, Y  +363.277, Z    +0.000, E1   +17.059, E3 +71852.409}
SPL {X  -165.638, Y  +376.493, Z    +0.000, E1    +4.395, E3 +71852.047}
SPL {X  -165.650, Y  +380.500, Z    +0.000, E1    +0.000, E3 +71851.157}
SPL {X  -165.650, Y  +381.832, Z    +0.000, E1    -2.686, E3 +71850.629}
SPL {X  -165.650, Y  +385.053, Z    +0.000, E1   -10.073, E3 +71850.535}
SPL {X  -165.650, Y  +388.847, Z    +0.000, E1   -19.524, E3 +71850.499}
SPL {X  -165.650, Y  +393.562, Z    +0.000, E1   -31.212, E3 +71849.983}
SPL {X  -165.650, Y  +400.090, Z    +0.000, E1   -44.561, E3 +71849.837}
SPL {X  -165.650, Y  +415.429, Z    +0.000, E1   -64.815, E3 +71847.896}
SPL {X  -165.650, Y  +470.008, Z    +0.000, E1   -77.011, E3 +71856.440}
SPL {X  -160.882, Y  +714.957, Z    +0.000, E1   -77.470, E3 +71940.146}
ENDSPLINE

SPLINE
SPL {X  -163.522, Y  +701.969, Z    +0.000, E1   -74.236, E3 +71969.802}
ENDSPLINE

SPLINE
SPL {X  -160.284, Y  +717.322, Z    +0.000, E1   -73.988, E3 +71981.135}
SPL {X  -156.453, Y  +729.928, Z    +0.000, E1   -73.507, E3 +71993.287}
SPL {X  -152.193, Y  +740.900, Z    +0.000, E1   -73.135, E3 +72002.853}
SPL {X  -148.880, Y  +748.126, Z    +0.000, E1   -72.716, E3 +72010.635}
SPL {X  -145.823, Y  +754.085, Z    +0.000, E1   -72.288, E3 +72017.406}
SPL {X  -141.906, Y  +760.955, Z    +0.000, E1   -72.057, E3 +72023.097}
SPL {X  -138.580, Y  +766.249, Z    +0.000, E1   -71.449, E3 +72030.186}
SPL {X  -134.851, Y  +771.704, Z    +0.000, E1   -71.081, E3 +72035.582}
SPL {X  -130.513, Y  +777.511, Z    +0.000, E1   -70.561, E3 +72041.764}
SPL {X  -127.002, Y  +781.850, Z    +0.000, E1   -69.819, E3 +72047.619}
SPL {X  -118.977, Y  +790.758, Z    +0.000, E1   -71.976, E3 +72043.736}
SPL {X   -54.135, Y  +832.054, Z    +0.000, E1   -56.519, E3 +72219.662}
ENDSPLINE

SPLINE
SPL {X  -119.915, Y  +789.781, Z    +0.000, E1   -62.637, E3 +72387.277}
SPL {X  -140.675, Y  +762.967, Z    +0.000, E1   -56.489, E3 +72387.619}
SPL {X  -155.138, Y  +733.569, Z    +0.000, E1   -46.550, E3 +72389.924}
SPL {X  -161.585, Y  +711.971, Z    +0.000, E1   -34.503, E3 +72388.974}
SPL {X  -164.796, Y  +692.295, Z    +0.000, E1   -19.289, E3 +72389.009}
SPL {X  -165.632, Y  +677.938, Z    +0.000, E1    -5.073, E3 +72388.380}
SPL {X  -165.650, Y  +673.297, Z    +0.000, E1    +0.232, E3 +72387.336}
SPL {X  -165.650, Y  +670.223, Z    +0.000, E1    +7.575, E3 +72386.817}
SPL {X  -165.650, Y  +666.568, Z    +0.000, E1   +16.799, E3 +72386.794}
SPL {X  -165.650, Y  +661.246, Z    +0.000, E1   +30.569, E3 +72386.574}
SPL {X  -165.650, Y  +655.398, Z    +0.000, E1   +43.871, E3 +72386.022}
SPL {X  -165.650, Y  +646.168, Z    +0.000, E1   +58.442, E3 +72385.117}
SPL {X  -165.650, Y  +629.125, Z    +0.000, E1   +72.389, E3 +72383.413}
SPL {X  -165.650, Y  +575.817, Z    +0.000, E1   +77.800, E3 +72394.731}
SPL {X  -161.405, Y  +341.238, Z    +0.000, E1   +76.606, E3 +72486.031}
SPL {X  -146.302, Y  +300.811, Z    +0.000, E1   +78.008, E3 +72487.148}
ENDSPLINE

SPLINE
SPL {X  -147.825, Y  +303.750, Z    +0.000, E1   +76.548, E3 +72501.580}
SPL {X  -148.167, Y  +304.430, Z    +0.000, E1   +75.276, E3 +72513.673}
ENDSPLINE

SPLINE
SPL {X  -146.983, Y  +302.107, Z    +0.000, E1   +74.473, E3 +72522.154}
SPL {X  -146.624, Y  +301.420, Z    +0.000, E1   +73.294, E3 +72532.638}
SPL {X  -144.830, Y  +298.101, Z    +0.000, E1   +72.333, E3 +72542.161}
SPL {X  -140.980, Y  +291.526, Z    +0.000, E1   +72.160, E3 +72547.086}
SPL {X  -137.379, Y  +285.943, Z    +0.000, E1   +71.537, E3 +72554.541}
SPL {X  -133.329, Y  +280.198, Z    +0.000, E1   +71.389, E3 +72558.570}
SPL {X  -130.835, Y  +276.902, Z    +0.000, E1   +70.642, E3 +72564.566}
SPL {X  -127.149, Y  +272.325, Z    +0.000, E1   +70.073, E3 +72569.817}
SPL {X  -123.924, Y  +268.578, Z    +0.000, E1   +70.633, E3 +72569.633}
SPL {X  -115.163, Y  +259.431, Z    +0.000, E1   +74.058, E3 +72560.743}
SPL {X   -55.479, Y  +222.417, Z    +0.000, E1   +56.403, E3 +72746.597}
ENDSPLINE

SPLINE
SPL {X  -130.757, Y  +276.802, Z    +0.000, E1   +58.343, E3 +72902.533}
SPL {X  -157.227, Y  +326.349, Z    +0.000, E1   +42.092, E3 +72906.179}
SPL {X  -163.771, Y  +353.623, Z    +0.000, E1   +25.144, E3 +72907.392}
SPL {X  -165.462, Y  +370.602, Z    +0.000, E1   +10.342, E3 +72906.342}
SPL {X  -165.650, Y  +380.417, Z    +0.000, E1    +0.167, E3 +72905.257}
SPL {X  -165.650, Y  +381.832, Z    +0.000, E1    -2.686, E3 +72904.683}
SPL {X  -165.650, Y  +385.053, Z    +0.000, E1   -10.073, E3 +72904.589}
SPL {X  -165.650, Y  +388.847, Z    +0.000, E1   -19.524, E3 +72904.553}
SPL {X  -165.650, Y  +393.562, Z    +0.000, E1   -31.212, E3 +72904.037}
SPL {X  -165.650, Y  +400.090, Z    +0.000, E1   -44.561, E3 +72903.892}
SPL {X  -165.650, Y  +415.429, Z    +0.000, E1   -64.815, E3 +72901.950}
SPL {X  -165.650, Y  +460.635, Z    +0.000, E1   -76.744, E3 +72907.847}
SPL {X  -165.650, Y  +476.745, Z    +0.000, E1   -77.150, E3 +72912.399}
SPL {X  -161.095, Y  +714.078, Z    +0.000, E1   -78.221, E3 +72986.029}
ENDSPLINE

SPLINE
SPL {X  -163.418, Y  +702.603, Z    +0.000, E1   -74.313, E3 +73023.425}
ENDSPLINE

SPLINE
SPL {X  -160.284, Y  +717.322, Z    +0.000, E1   -73.988, E3 +73035.189}
SPL {X  -157.512, Y  +726.783, Z    +0.000, E1   -73.653, E3 +73043.903}
SPL {X  -155.383, Y  +732.911, Z    +0.000, E1   -73.297, E3 +73050.829}
SPL {X  -152.193, Y  +740.900, Z    +0.000, E1   -73.135, E3 +73056.907}
SPL {X  -148.880, Y  +748.126, Z    +0.000, E1   -72.716, E3 +73064.689}
SPL {X  -145.823, Y  +754.085, Z    +0.000, E1   -72.288, E3 +73071.460}
SPL {X  -141.906, Y  +760.955, Z    +0.000, E1   -72.057, E3 +73077.151}
SPL {X  -138.580, Y  +766.249, Z    +0.000, E1   -71.449, E3 +73084.240}
SPL {X  -134.851, Y  +771.704, Z    +0.000, E1   -71.081, E3 +73089.636}
SPL {X  -130.513, Y  +777.511, Z    +0.000, E1   -70.561, E3 +73095.818}
SPL {X  -127.002, Y  +781.850, Z    +0.000, E1   -69.819, E3 +73101.673}
SPL {X  -118.977, Y  +790.758, Z    +0.000, E1   -71.976, E3 +73097.790}
SPL {X   -54.135, Y  +832.054, Z    +0.000, E1   -56.519, E3 +73273.716}
ENDSPLINE

SPLINE
SPL {X  -119.915, Y  +789.781, Z    +0.000, E1   -62.637, E3 +73441.331}
SPL {X  -140.675, Y  +762.967, Z    +0.000, E1   -56.489, E3 +73441.673}
SPL {X  -155.138, Y  +733.569, Z    +0.000, E1   -46.550, E3 +73443.978}
SPL {X  -161.585, Y  +711.971, Z    +0.000, E1   -34.503, E3 +73443.028}
SPL {X  -164.796, Y  +692.295, Z    +0.000, E1   -19.289, E3 +73443.063}
SPL {X  -165.632, Y  +677.938, Z    +0.000, E1    -5.073, E3 +73442.434}
SPL {X  -165.650, Y  +673.297, Z    +0.000, E1    +0.232, E3 +73441.390}
SPL {X  -165.650, Y  +670.223, Z    +0.000, E1    +7.575, E3 +73440.871}
SPL {X  -165.650, Y  +666.568, Z    +0.000, E1   +16.799, E3 +73440.848}
SPL {X  -165.650, Y  +661.246, Z    +0.000, E1   +30.569, E3 +73440.628}
SPL {X  -165.650, Y  +655.398, Z    +0.000, E1   +43.871, E3 +73440.076}
SPL {X  -165.650, Y  +646.168, Z    +0.000, E1   +58.442, E3 +73439.171}
SPL {X  -165.650, Y  +629.125, Z    +0.000, E1   +72.389, E3 +73437.467}
SPL {X  -165.650, Y  +575.817, Z    +0.000, E1   +77.800, E3 +73448.785}
SPL {X  -161.405, Y  +341.238, Z    +0.000, E1   +76.606, E3 +73540.085}
SPL {X  -146.302, Y  +300.811, Z    +0.000, E1   +78.008, E3 +73541.202}
ENDSPLINE

SPLINE
SPL {X  -147.825, Y  +303.750, Z    +0.000, E1   +76.548, E3 +73555.634}
SPL {X  -148.167, Y  +304.430, Z    +0.000, E1   +75.276, E3 +73567.727}
ENDSPLINE

SPLINE
SPL {X  -146.983, Y  +302.107, Z    +0.000, E1   +74.473, E3 +73576.208}
SPL {X  -146.624, Y  +301.420, Z    +0.000, E1   +73.294, E3 +73586.692}
SPL {X  -144.830, Y  +298.101, Z    +0.000, E1   +72.333, E3 +73596.215}
SPL {X  -140.980, Y  +291.526, Z    +0.000, E1   +72.160, E3 +73601.140}
SPL {X  -137.379, Y  +285.943, Z    +0.000, E1   +71.537, E3 +73608.595}
SPL {X  -133.329, Y  +280.198, Z    +0.000, E1   +71.389, E3 +73612.624}
SPL {X  -130.835, Y  +276.902, Z    +0.000, E1   +70.642, E3 +73618.620}
SPL {X  -127.149, Y  +272.325, Z    +0.000, E1   +70.073, E3 +73623.871}
SPL {X  -123.924, Y  +268.578, Z    +0.000, E1   +70.633, E3 +73623.687}
SPL {X  -115.163, Y  +259.431, Z    +0.000, E1   +74.058, E3 +73614.797}
SPL {X   -55.479, Y  +222.417, Z    +0.000, E1   +56.403, E3 +73800.651}
ENDSPLINE

SPLINE
SPL {X  -130.757, Y  +276.802, Z    +0.000, E1   +58.343, E3 +73956.587}
SPL {X  -157.227, Y  +326.349, Z    +0.000, E1   +42.092, E3 +73960.233}
SPL {X  -163.771, Y  +353.623, Z    +0.000, E1   +25.144, E3 +73961.446}
SPL {X  -165.171, Y  +365.918, Z    +0.000, E1   +14.637, E3 +73960.660}
SPL {X  -165.638, Y  +376.493, Z    +0.000, E1    +4.395, E3 +73960.155}
SPL {X  -165.650, Y  +380.829, Z    +0.000, E1    -0.360, E3 +73959.135}
SPL {X  -165.650, Y  +385.053, Z    +0.000, E1   -10.073, E3 +73958.643}
SPL {X  -165.650, Y  +388.847, Z    +0.000, E1   -19.524, E3 +73958.607}
SPL {X  -165.650, Y  +393.562, Z    +0.000, E1   -31.212, E3 +73958.091}
SPL {X  -165.650, Y  +400.090, Z    +0.000, E1   -44.561, E3 +73957.946}
SPL {X  -165.650, Y  +415.429, Z    +0.000, E1   -64.815, E3 +73956.004}
SPL {X  -165.650, Y  +470.008, Z    +0.000, E1   -77.011, E3 +73964.548}
SPL {X  -160.882, Y  +714.957, Z    +0.000, E1   -77.470, E3 +74048.254}
ENDSPLINE

SPLINE
SPL {X  -164.302, Y  +696.586, Z    +0.000, E1   -74.218, E3 +74074.916}
ENDSPLINE

SPLINE
SPL {X  -160.977, Y  +714.570, Z    +0.000, E1   -74.086, E3 +74086.828}
SPL {X  -156.453, Y  +729.928, Z    +0.000, E1   -73.507, E3 +74101.395}
SPL {X  -152.193, Y  +740.900, Z    +0.000, E1   -73.135, E3 +74110.961}
SPL {X  -148.880, Y  +748.126, Z    +0.000, E1   -72.716, E3 +74118.743}
SPL {X  -145.823, Y  +754.085, Z    +0.000, E1   -72.288, E3 +74125.514}
SPL {X  -141.906, Y  +760.955, Z    +0.000, E1   -72.057, E3 +74131.205}
SPL {X  -138.580, Y  +766.249, Z    +0.000, E1   -71.449, E3 +74138.295}
SPL {X  -134.851, Y  +771.704, Z    +0.000, E1   -71.081, E3 +74143.690}
SPL {X  -130.513, Y  +777.511, Z    +0.000, E1   -70.561, E3 +74149.872}
SPL {X  -127.002, Y  +781.850, Z    +0.000, E1   -69.819, E3 +74155.727}
SPL {X  -118.977, Y  +790.758, Z    +0.000, E1   -71.976, E3 +74151.844}
SPL {X   -54.135, Y  +832.054, Z    +0.000, E1   -56.519, E3 +74327.770}
ENDSPLINE

SPLINE
SPL {X  -119.915, Y  +789.781, Z    +0.000, E1   -62.637, E3 +74495.385}
SPL {X  -140.675, Y  +762.967, Z    +0.000, E1   -56.489, E3 +74495.727}
SPL {X  -155.138, Y  +733.569, Z    +0.000, E1   -46.550, E3 +74498.032}
SPL {X  -161.585, Y  +711.971, Z    +0.000, E1   -34.503, E3 +74497.082}
SPL {X  -164.796, Y  +692.295, Z    +0.000, E1   -19.289, E3 +74497.117}
SPL {X  -165.632, Y  +677.938, Z    +0.000, E1    -5.073, E3 +74496.488}
SPL {X  -165.650, Y  +673.297, Z    +0.000, E1    +0.232, E3 +74495.444}
SPL {X  -165.650, Y  +670.223, Z    +0.000, E1    +7.575, E3 +74494.925}
SPL {X  -165.650, Y  +666.568, Z    +0.000, E1   +16.799, E3 +74494.902}
SPL {X  -165.650, Y  +661.246, Z    +0.000, E1   +30.569, E3 +74494.682}
SPL {X  -165.650, Y  +655.398, Z    +0.000, E1   +43.871, E3 +74494.130}
SPL {X  -165.650, Y  +646.168, Z    +0.000, E1   +58.442, E3 +74493.225}
SPL {X  -165.650, Y  +629.125, Z    +0.000, E1   +72.389, E3 +74491.521}
SPL {X  -165.650, Y  +575.817, Z    +0.000, E1   +77.800, E3 +74502.839}
SPL {X  -161.405, Y  +341.238, Z    +0.000, E1   +76.606, E3 +74594.139}
SPL {X  -146.302, Y  +300.811, Z    +0.000, E1   +78.008, E3 +74595.256}
ENDSPLINE

SPLINE
SPL {X  -147.825, Y  +303.750, Z    +0.000, E1   +76.548, E3 +74609.688}
SPL {X  -148.167, Y  +304.430, Z    +0.000, E1   +75.276, E3 +74621.781}
ENDSPLINE

SPLINE
SPL {X  -146.983, Y  +302.107, Z    +0.000, E1   +74.473, E3 +74630.262}
SPL {X  -146.624, Y  +301.420, Z    +0.000, E1   +73.294, E3 +74640.746}
SPL {X  -144.830, Y  +298.101, Z    +0.000, E1   +72.333, E3 +74650.269}
SPL {X  -140.980, Y  +291.526, Z    +0.000, E1   +72.160, E3 +74655.194}
SPL {X  -137.379, Y  +285.943, Z    +0.000, E1   +71.537, E3 +74662.649}
SPL {X  -133.329, Y  +280.198, Z    +0.000, E1   +71.389, E3 +74666.678}
SPL {X  -130.835, Y  +276.902, Z    +0.000, E1   +70.642, E3 +74672.674}
SPL {X  -127.149, Y  +272.325, Z    +0.000, E1   +70.073, E3 +74677.925}
SPL {X  -123.924, Y  +268.578, Z    +0.000, E1   +70.633, E3 +74677.741}
SPL {X  -115.163, Y  +259.431, Z    +0.000, E1   +74.058, E3 +74668.851}
SPL {X   -55.479, Y  +222.417, Z    +0.000, E1   +56.403, E3 +74854.705}
ENDSPLINE

SPLINE
SPL {X  -130.757, Y  +276.802, Z    +0.000, E1   +58.343, E3 +75010.641}
SPL {X  -157.227, Y  +326.349, Z    +0.000, E1   +42.092, E3 +75014.287}
SPL {X  -163.771, Y  +353.623, Z    +0.000, E1   +25.144, E3 +75015.500}
SPL {X  -165.462, Y  +370.602, Z    +0.000, E1   +10.342, E3 +75014.450}
SPL {X  -165.650, Y  +380.417, Z    +0.000, E1    +0.167, E3 +75013.365}
SPL {X  -165.650, Y  +381.832, Z    +0.000, E1    -2.686, E3 +75012.791}
SPL {X  -165.650, Y  +385.053, Z    +0.000, E1   -10.073, E3 +75012.697}
SPL {X  -165.650, Y  +388.847, Z    +0.000, E1   -19.524, E3 +75012.661}
SPL {X  -165.650, Y  +393.562, Z    +0.000, E1   -31.212, E3 +75012.145}
SPL {X  -165.650, Y  +400.090, Z    +0.000, E1   -44.561, E3 +75012.000}
SPL {X  -165.650, Y  +415.429, Z    +0.000, E1   -64.815, E3 +75010.058}
SPL {X  -165.650, Y  +460.635, Z    +0.000, E1   -76.744, E3 +75015.955}
SPL {X  -165.650, Y  +476.745, Z    +0.000, E1   -77.150, E3 +75020.507}
SPL {X  -161.095, Y  +714.078, Z    +0.000, E1   -78.221, E3 +75094.138}
ENDSPLINE

SPLINE
SPL {X  -163.418, Y  +702.603, Z    +0.000, E1   -74.313, E3 +75131.533}
ENDSPLINE

SPLINE
SPL {X  -160.284, Y  +717.322, Z    +0.000, E1   -73.988, E3 +75143.297}
SPL {X  -157.512, Y  +726.783, Z    +0.000, E1   -73.653, E3 +75152.011}
SPL {X  -155.383, Y  +732.911, Z    +0.000, E1   -73.297, E3 +75158.937}
SPL {X  -152.193, Y  +740.900, Z    +0.000, E1   -73.135, E3 +75165.015}
SPL {X  -148.880, Y  +748.126, Z    +0.000, E1   -72.716, E3 +75172.797}
SPL {X  -145.823, Y  +754.085, Z    +0.000, E1   -72.288, E3 +75179.568}
SPL {X  -141.906, Y  +760.955, Z    +0.000, E1   -72.057, E3 +75185.259}
SPL {X  -138.580, Y  +766.249, Z    +0.000, E1   -71.449, E3 +75192.349}
SPL {X  -134.851, Y  +771.704, Z    +0.000, E1   -71.081, E3 +75197.744}
SPL {X  -130.513, Y  +777.511, Z    +0.000, E1   -70.561, E3 +75203.926}
SPL {X  -127.002, Y  +781.850, Z    +0.000, E1   -69.819, E3 +75209.781}
SPL {X  -118.977, Y  +790.758, Z    +0.000, E1   -71.976, E3 +75205.898}
SPL {X   -54.135, Y  +832.054, Z    +0.000, E1   -56.519, E3 +75381.824}
ENDSPLINE

SPLINE
SPL {X  -119.915, Y  +789.781, Z    +0.000, E1   -62.637, E3 +75549.439}
SPL {X  -140.675, Y  +762.967, Z    +0.000, E1   -56.489, E3 +75549.781}
SPL {X  -155.138, Y  +733.569, Z    +0.000, E1   -46.550, E3 +75552.086}
SPL {X  -161.585, Y  +711.971, Z    +0.000, E1   -34.503, E3 +75551.136}
SPL {X  -164.796, Y  +692.295, Z    +0.000, E1   -19.289, E3 +75551.171}
SPL {X  -165.632, Y  +677.938, Z    +0.000, E1    -5.073, E3 +75550.542}
SPL {X  -165.650, Y  +673.297, Z    +0.000, E1    +0.232, E3 +75549.498}
SPL {X  -165.650, Y  +670.223, Z    +0.000, E1    +7.575, E3 +75548.979}
SPL {X  -165.650, Y  +666.568, Z    +0.000, E1   +16.799, E3 +75548.956}
SPL {X  -165.650, Y  +661.246, Z    +0.000, E1   +30.569, E3 +75548.736}
SPL {X  -165.650, Y  +655.398, Z    +0.000, E1   +43.871, E3 +75548.184}
SPL {X  -165.650, Y  +646.168, Z    +0.000, E1   +58.442, E3 +75547.279}
SPL {X  -165.650, Y  +629.125, Z    +0.000, E1   +72.389, E3 +75545.575}
SPL {X  -165.650, Y  +575.817, Z    +0.000, E1   +77.800, E3 +75556.893}
SPL {X  -161.405, Y  +341.238, Z    +0.000, E1   +76.606, E3 +75648.193}
SPL {X  -146.302, Y  +300.811, Z    +0.000, E1   +78.008, E3 +75649.310}
ENDSPLINE

SPLINE
SPL {X  -147.825, Y  +303.750, Z    +0.000, E1   +76.548, E3 +75663.742}
SPL {X  -148.167, Y  +304.430, Z    +0.000, E1   +75.276, E3 +75675.835}
ENDSPLINE

SPLINE
SPL {X  -146.983, Y  +302.107, Z    +0.000, E1   +74.473, E3 +75684.316}
SPL {X  -146.624, Y  +301.420, Z    +0.000, E1   +73.294, E3 +75694.800}
SPL {X  -144.830, Y  +298.101, Z    +0.000, E1   +72.333, E3 +75704.323}
SPL {X  -140.980, Y  +291.526, Z    +0.000, E1   +72.160, E3 +75709.249}
SPL {X  -137.379, Y  +285.943, Z    +0.000, E1   +71.537, E3 +75716.703}
SPL {X  -133.329, Y  +280.198, Z    +0.000, E1   +71.389, E3 +75720.732}
SPL {X  -130.835, Y  +276.902, Z    +0.000, E1   +70.642, E3 +75726.728}
SPL {X  -127.149, Y  +272.325, Z    +0.000, E1   +70.073, E3 +75731.979}
SPL {X  -123.924, Y  +268.578, Z    +0.000, E1   +70.633, E3 +75731.795}
SPL {X  -115.163, Y  +259.431, Z    +0.000, E1   +74.058, E3 +75722.905}
SPL {X   -55.479, Y  +222.417, Z    +0.000, E1   +56.403, E3 +75908.759}
ENDSPLINE

SPLINE
SPL {X  -130.757, Y  +276.802, Z    +0.000, E1   +58.343, E3 +76064.695}
SPL {X  -157.227, Y  +326.349, Z    +0.000, E1   +42.092, E3 +76068.341}
SPL {X  -163.771, Y  +353.623, Z    +0.000, E1   +25.144, E3 +76069.554}
SPL {X  -165.462, Y  +370.602, Z    +0.000, E1   +10.342, E3 +76068.504}
SPL {X  -165.650, Y  +380.417, Z    +0.000, E1    +0.167, E3 +76067.419}
SPL {X  -165.650, Y  +381.832, Z    +0.000, E1    -2.686, E3 +76066.845}
SPL {X  -165.650, Y  +385.053, Z    +0.000, E1   -10.073, E3 +76066.751}
SPL {X  -165.650, Y  +388.847, Z    +0.000, E1   -19.524, E3 +76066.715}
SPL {X  -165.650, Y  +394.451, Z    +0.000, E1   -33.170, E3 +76066.128}
SPL {X  -165.650, Y  +401.692, Z    +0.000, E1   -47.300, E3 +76066.111}
SPL {X  -165.650, Y  +415.429, Z    +0.000, E1   -64.815, E3 +76064.112}
SPL {X  -165.650, Y  +470.008, Z    +0.000, E1   -77.011, E3 +76072.656}
SPL {X  -160.882, Y  +714.957, Z    +0.000, E1   -77.470, E3 +76156.362}
ENDSPLINE

SPLINE
SPL {X  -164.302, Y  +696.586, Z    +0.000, E1   -74.218, E3 +76183.024}
ENDSPLINE

SPLINE
SPL {X  -160.977, Y  +714.570, Z    +0.000, E1   -74.086, E3 +76194.936}
SPL {X  -156.453, Y  +729.928, Z    +0.000, E1   -73.507, E3 +76209.503}
SPL {X  -152.193, Y  +740.900, Z    +0.000, E1   -73.135, E3 +76219.069}
SPL {X  -148.880, Y  +748.126, Z    +0.000, E1   -72.716, E3 +76226.851}
SPL {X  -144.434, Y  +756.610, Z    +0.000, E1   -72.338, E3 +76234.701}
SPL {X  -141.532, Y  +761.573, Z    +0.000, E1   -71.800, E3 +76241.341}
SPL {X  -138.580, Y  +766.249, Z    +0.000, E1   -71.449, E3 +76246.403}
SPL {X  -134.851, Y  +771.704, Z    +0.000, E1   -71.081, E3 +76251.798}
SPL {X  -131.668, Y  +776.015, Z    +0.000, E1   -70.566, E3 +76257.071}
SPL {X  -128.114, Y  +780.508, Z    +0.000, E1   -70.155, E3 +76261.667}
SPL {X  -123.825, Y  +785.533, Z    +0.000, E1   -70.642, E3 +76262.415}
SPL {X  -111.068, Y  +798.397, Z    +0.000, E1   -72.944, E3 +76259.859}
SPL {X   -54.368, Y  +831.974, Z    +0.000, E1   -57.152, E3 +76411.742}
ENDSPLINE

SPLINE
SPL {X  -111.514, Y  +797.993, Z    +0.000, E1   -63.064, E3 +76597.873}
SPL {X  -140.675, Y  +762.967, Z    +0.000, E1   -56.489, E3 +76603.836}
SPL {X  -155.138, Y  +733.569, Z    +0.000, E1   -46.550, E3 +76606.140}
SPL {X  -162.699, Y  +706.626, Z    +0.000, E1   -30.890, E3 +76605.182}
SPL {X  -165.420, Y  +684.230, Z    +0.000, E1   -11.665, E3 +76604.933}
SPL {X  -165.650, Y  +673.591, Z    +0.000, E1    -0.194, E3 +76603.676}
SPL {X  -165.650, Y  +671.349, Z    +0.000, E1    +4.619, E3 +76603.134}
SPL {X  -165.650, Y  +666.568, Z    +0.000, E1   +16.799, E3 +76603.010}
SPL {X  -165.650, Y  +661.246, Z    +0.000, E1   +30.569, E3 +76602.790}
SPL {X  -165.650, Y  +655.398, Z    +0.000, E1   +43.871, E3 +76602.238}
SPL {X  -165.650, Y  +646.168, Z    +0.000, E1   +58.442, E3 +76601.333}
SPL {X  -165.650, Y  +629.125, Z    +0.000, E1   +72.389, E3 +76599.629}
SPL {X  -165.650, Y  +575.817, Z    +0.000, E1   +77.800, E3 +76610.947}
SPL {X  -161.405, Y  +341.238, Z    +0.000, E1   +76.606, E3 +76702.247}
SPL {X  -146.302, Y  +300.811, Z    +0.000, E1   +78.008, E3 +76703.364}
ENDSPLINE

SPLINE
SPL {X  -147.825, Y  +303.750, Z    +0.000, E1   +76.548, E3 +76717.796}
SPL {X  -148.167, Y  +304.430, Z    +0.000, E1   +75.276, E3 +76729.889}
ENDSPLINE

SPLINE
SPL {X  -146.983, Y  +302.107, Z    +0.000, E1   +74.473, E3 +76738.370}
SPL {X  -146.624, Y  +301.420, Z    +0.000, E1   +73.294, E3 +76748.854}
SPL {X  -144.830, Y  +298.101, Z    +0.000, E1   +72.333, E3 +76758.377}
SPL {X  -140.980, Y  +291.526, Z    +0.000, E1   +72.160, E3 +76763.303}
SPL {X  -137.379, Y  +285.943, Z    +0.000, E1   +71.537, E3 +76770.757}
SPL {X  -133.329, Y  +280.198, Z    +0.000, E1   +71.389, E3 +76774.786}
SPL {X  -130.835, Y  +276.902, Z    +0.000, E1   +70.642, E3 +76780.782}
SPL {X  -127.149, Y  +272.325, Z    +0.000, E1   +70.073, E3 +76786.033}
SPL {X  -123.924, Y  +268.578, Z    +0.000, E1   +70.633, E3 +76785.849}
SPL {X  -115.163, Y  +259.431, Z    +0.000, E1   +74.058, E3 +76776.959}
SPL {X   -55.479, Y  +222.417, Z    +0.000, E1   +56.403, E3 +76962.813}
ENDSPLINE

SPLINE
SPL {X  -130.757, Y  +276.802, Z    +0.000, E1   +58.343, E3 +77118.749}
SPL {X  -154.788, Y  +319.502, Z    +0.000, E1   +45.389, E3 +77122.948}
SPL {X  -161.887, Y  +343.393, Z    +0.000, E1   +32.461, E3 +77123.404}
SPL {X  -164.949, Y  +363.277, Z    +0.000, E1   +17.059, E3 +77122.679}
SPL {X  -165.638, Y  +376.493, Z    +0.000, E1    +4.395, E3 +77122.317}
SPL {X  -165.650, Y  +380.500, Z    +0.000, E1    +0.000, E3 +77121.427}
SPL {X  -165.650, Y  +381.832, Z    +0.000, E1    -2.686, E3 +77120.900}
SPL {X  -165.650, Y  +385.053, Z    +0.000, E1   -10.073, E3 +77120.805}
SPL {X  -165.650, Y  +388.847, Z    +0.000, E1   -19.524, E3 +77120.769}
SPL {X  -165.650, Y  +393.562, Z    +0.000, E1   -31.212, E3 +77120.253}
SPL {X  -165.650, Y  +400.090, Z    +0.000, E1   -44.561, E3 +77120.108}
SPL {X  -165.650, Y  +415.429, Z    +0.000, E1   -64.815, E3 +77118.166}
SPL {X  -165.650, Y  +470.008, Z    +0.000, E1   -77.011, E3 +77126.710}
SPL {X  -160.882, Y  +714.957, Z    +0.000, E1   -77.470, E3 +77210.416}
ENDSPLINE

SPLINE
SPL {X  -164.302, Y  +696.586, Z    +0.000, E1   -74.218, E3 +77237.078}
ENDSPLINE

SPLINE
SPL {X  -160.977, Y  +714.570, Z    +0.000, E1   -74.086, E3 +77248.990}
SPL {X  -156.453, Y  +729.928, Z    +0.000, E1   -73.507, E3 +77263.557}
SPL {X  -152.193, Y  +740.900, Z    +0.000, E1   -73.135, E3 +77273.123}
SPL {X  -148.880, Y  +748.126, Z    +0.000, E1   -72.716, E3 +77280.905}
SPL {X  -145.823, Y  +754.085, Z    +0.000, E1   -72.288, E3 +77287.676}
SPL {X  -141.906, Y  +760.955, Z    +0.000, E1   -72.057, E3 +77293.367}
SPL {X  -138.580, Y  +766.249, Z    +0.000, E1   -71.449, E3 +77300.457}
SPL {X  -134.851, Y  +771.704, Z    +0.000, E1   -71.081, E3 +77305.852}
SPL {X  -130.513, Y  +777.511, Z    +0.000, E1   -70.561, E3 +77312.034}
SPL {X  -127.002, Y  +781.850, Z    +0.000, E1   -69.819, E3 +77317.889}
SPL {X  -118.977, Y  +790.758, Z    +0.000, E1   -71.976, E3 +77314.007}
SPL {X   -54.135, Y  +832.054, Z    +0.000, E1   -56.519, E3 +77489.932}
ENDSPLINE

SPLINE
SPL {X  -119.915, Y  +789.781, Z    +0.000, E1   -62.637, E3 +77657.547}
SPL {X  -140.675, Y  +762.967, Z    +0.000, E1   -56.489, E3 +77657.890}
SPL {X  -155.138, Y  +733.569, Z    +0.000, E1   -46.550, E3 +77660.194}
SPL {X  -161.585, Y  +711.971, Z    +0.000, E1   -34.503, E3 +77659.244}
SPL {X  -164.796, Y  +692.295, Z    +0.000, E1   -19.289, E3 +77659.279}
SPL {X  -165.632, Y  +677.938, Z    +0.000, E1    -5.073, E3 +77658.650}
SPL {X  -165.650, Y  +673.297, Z    +0.000, E1    +0.232, E3 +77657.607}
SPL {X  -165.650, Y  +670.223, Z    +0.000, E1    +7.575, E3 +77657.087}
SPL {X  -165.650, Y  +666.568, Z    +0.000, E1   +16.799, E3 +77657.064}
SPL {X  -165.650, Y  +661.246, Z    +0.000, E1   +30.569, E3 +77656.844}
SPL {X  -165.650, Y  +655.398, Z    +0.000, E1   +43.871, E3 +77656.292}
SPL {X  -165.650, Y  +646.168, Z    +0.000, E1   +58.442, E3 +77655.387}
SPL {X  -165.650, Y  +629.125, Z    +0.000, E1   +72.389, E3 +77653.683}
SPL {X  -165.650, Y  +575.817, Z    +0.000, E1   +77.800, E3 +77665.001}
SPL {X  -161.405, Y  +341.238, Z    +0.000, E1   +76.606, E3 +77756.301}
SPL {X  -146.302, Y  +300.811, Z    +0.000, E1   +78.008, E3 +77757.418}
ENDSPLINE

SPLINE
SPL {X  -147.825, Y  +303.750, Z    +0.000, E1   +76.548, E3 +77771.850}
SPL {X  -148.167, Y  +304.430, Z    +0.000, E1   +75.276, E3 +77783.943}
ENDSPLINE

SPLINE
SPL {X  -146.983, Y  +302.107, Z    +0.000, E1   +74.473, E3 +77792.424}
SPL {X  -146.624, Y  +301.420, Z    +0.000, E1   +73.294, E3 +77802.908}
SPL {X  -144.830, Y  +298.101, Z    +0.000, E1   +72.333, E3 +77812.431}
SPL {X  -140.980, Y  +291.526, Z    +0.000, E1   +72.160, E3 +77817.357}
SPL {X  -137.379, Y  +285.943, Z    +0.000, E1   +71.537, E3 +77824.811}
SPL {X  -132.604, Y  +279.221, Z    +0.000, E1   +70.988, E3 +77831.783}
SPL {X  -129.663, Y  +275.410, Z    +0.000, E1   +70.632, E3 +77835.707}
SPL {X  -127.149, Y  +272.325, Z    +0.000, E1   +70.073, E3 +77840.087}
SPL {X  -123.924, Y  +268.578, Z    +0.000, E1   +70.633, E3 +77839.904}
SPL {X  -115.163, Y  +259.431, Z    +0.000, E1   +74.058, E3 +77831.013}
SPL {X   -55.479, Y  +222.417, Z    +0.000, E1   +56.403, E3 +78016.867}
ENDSPLINE

SPLINE
SPL {X  -130.757, Y  +276.802, Z    +0.000, E1   +58.343, E3 +78172.803}
SPL {X  -157.227, Y  +326.349, Z    +0.000, E1   +42.092, E3 +78176.449}
SPL {X  -163.771, Y  +353.623, Z    +0.000, E1   +25.144, E3 +78177.662}
SPL {X  -165.171, Y  +365.918, Z    +0.000, E1   +14.637, E3 +78176.876}
SPL {X  -165.638, Y  +376.493, Z    +0.000, E1    +4.395, E3 +78176.371}
SPL {X  -165.650, Y  +380.829, Z    +0.000, E1    -0.360, E3 +78175.351}
SPL {X  -165.650, Y  +385.053, Z    +0.000, E1   -10.073, E3 +78174.859}
SPL {X  -165.650, Y  +388.847, Z    +0.000, E1   -19.524, E3 +78174.823}
SPL {X  -165.650, Y  +393.562, Z    +0.000, E1   -31.212, E3 +78174.307}
SPL {X  -165.650, Y  +400.090, Z    +0.000, E1   -44.561, E3 +78174.162}
SPL {X  -165.650, Y  +415.429, Z    +0.000, E1   -64.815, E3 +78172.220}
SPL {X  -165.650, Y  +470.008, Z    +0.000, E1   -77.011, E3 +78180.764}
SPL {X  -161.095, Y  +714.078, Z    +0.000, E1   -78.221, E3 +78256.300}
ENDSPLINE

SPLINE
SPL {X  -163.418, Y  +702.603, Z    +0.000, E1   -74.313, E3 +78293.695}
ENDSPLINE

SPLINE
SPL {X  -160.284, Y  +717.322, Z    +0.000, E1   -73.988, E3 +78305.459}
SPL {X  -157.512, Y  +726.783, Z    +0.000, E1   -73.653, E3 +78314.173}
SPL {X  -155.383, Y  +732.911, Z    +0.000, E1   -73.297, E3 +78321.100}
SPL {X  -152.193, Y  +740.900, Z    +0.000, E1   -73.135, E3 +78327.178}
SPL {X  -148.880, Y  +748.126, Z    +0.000, E1   -72.716, E3 +78334.959}
SPL {X  -144.434, Y  +756.610, Z    +0.000, E1   -72.338, E3 +78342.809}
SPL {X  -141.532, Y  +761.573, Z    +0.000, E1   -71.800, E3 +78349.449}
SPL {X  -138.580, Y  +766.249, Z    +0.000, E1   -71.449, E3 +78354.511}
SPL {X  -134.851, Y  +771.704, Z    +0.000, E1   -71.081, E3 +78359.906}
SPL {X  -131.668, Y  +776.015, Z    +0.000, E1   -70.566, E3 +78365.180}
SPL {X  -128.114, Y  +780.508, Z    +0.000, E1   -70.155, E3 +78369.775}
SPL {X  -123.825, Y  +785.533, Z    +0.000, E1   -70.642, E3 +78370.523}
SPL {X  -111.068, Y  +798.397, Z    +0.000, E1   -72.944, E3 +78367.967}
SPL {X   -54.368, Y  +831.974, Z    +0.000, E1   -57.152, E3 +78519.850}
ENDSPLINE

SPLINE
SPL {X  -111.514, Y  +797.993, Z    +0.000, E1   -63.064, E3 +78705.981}
SPL {X  -140.675, Y  +762.967, Z    +0.000, E1   -56.489, E3 +78711.944}
SPL {X  -155.138, Y  +733.569, Z    +0.000, E1   -46.550, E3 +78714.248}
SPL {X  -161.585, Y  +711.971, Z    +0.000, E1   -34.503, E3 +78713.298}
SPL {X  -164.796, Y  +692.295, Z    +0.000, E1   -19.289, E3 +78713.333}
SPL {X  -165.632, Y  +677.938, Z    +0.000, E1    -5.073, E3 +78712.704}
SPL {X  -165.650, Y  +673.500, Z    +0.000, E1    +0.000, E3 +78711.738}
SPL {X  -165.650, Y  +671.349, Z    +0.000, E1    +4.619, E3 +78711.243}
SPL {X  -165.650, Y  +666.568, Z    +0.000, E1   +16.799, E3 +78711.118}
SPL {X  -165.650, Y  +661.246, Z    +0.000, E1   +30.569, E3 +78710.898}
SPL {X  -165.650, Y  +655.398, Z    +0.000, E1   +43.871, E3 +78710.346}
SPL {X  -165.650, Y  +646.168, Z    +0.000, E1   +58.442, E3 +78709.441}
SPL {X  -165.650, Y  +629.125, Z    +0.000, E1   +72.389, E3 +78707.738}
SPL {X  -165.650, Y  +575.817, Z    +0.000, E1   +77.800, E3 +78719.056}
SPL {X  -161.405, Y  +341.238, Z    +0.000, E1   +76.606, E3 +78810.355}
SPL {X  -145.880, Y  +300.022, Z    +0.000, E1   +78.339, E3 +78807.894}
ENDSPLINE

SPLINE
SPL {X  -146.769, Y  +301.697, Z    +0.000, E1   +77.642, E3 +78814.947}
SPL {X  -147.825, Y  +303.750, Z    +0.000, E1   +76.548, E3 +78825.904}
SPL {X  -148.167, Y  +304.430, Z    +0.000, E1   +75.276, E3 +78837.997}
ENDSPLINE

